// no rotation
IF ABS(angle)<g_smallAng THEN
	angle :=0;
	axis[1]:=1;
	axis[2]:=0;
	axis[3]:=0;
// rotate pi
ELSIF ABS(angle-pi)< g_smallAng THEN
	angle :=PI;
	axis[1]:=SQRT((LIMIT(-1, rot[1,1],1)+1)/2);
	axis[2]:=SQRT((LIMIT(-1, rot[2,2],1)+1)/2);
	axis[3]:=SQRT((limit(-1, rot[3,3],1)+1)/2);
	IF axis[1]>g_smallNum THEN
		axis[2]:=0.5*rot[1,2]/axis[1];
		axis[3]:=0.5*rot[1,3]/axis[1];
	ELSIF axis[2]>g_smallNum THEN
		axis[1]:=0.5*rot[2,1]/axis[2];
		axis[3]:=0.5*rot[2,3]/axis[2];
	ELSE
		axis[1]:=0.5*rot[3,1]/axis[3];
		axis[2]:=0.5*rot[3,2]/axis[3];
	END_IF
// others
ELSE
	tmp:=2*SIN(angle);
	axis[1]:=(rot[3,2]-rot[2,3])/tmp;
	axis[2]:=(rot[1,3]-rot[3,1])/tmp;
	axis[3]:=(rot[2,1]-rot[1,2])/tmp;
END_IF

// normalize
normalize(axis);

END_FUNCTION

// ---- AgiMaths/MatrixLib/normalize.TcPOU
// normalize the input vector
FUNCTION normalize : bool
VAR_IN_OUT
	vec :ARRAY[*] OF LREAL;
END_VAR
VAR
	m,i:DINT;
	vecNorm :LREAL;
END_VAR

m:=UPPER_BOUND(vec,1);
vecNorm :=norm(vec);

// if vector close to zero, remain the same;
IF vecNorm< g_smallNum THEN
	normalize :=FALSE;
	RETURN;
END_IF

FOR i:=1 TO m DO
	vec[i] := vec[i]/vecNorm;
END_FOR
normalize :=TRUE;

END_FUNCTION

// ---- AgiMaths/MatrixLib/norm.TcPOU
// return the norm of a vector
FUNCTION norm : LREAL
VAR_IN_OUT CONSTANT
	vec :ARRAY[*] OF LREAL;
END_VAR
VAR
	m,i:DINT;
END_VAR

m:=UPPER_BOUND(vec,1);
norm:=0;
FOR i:=1 TO m DO
	norm := norm + vec[i]*vec[i];
END_FOR

norm := SQRT(norm);

END_FUNCTION

// ---- AgiMaths/MatrixLib/vecMultiNum.TcPOU
// vecB=VecA*num
FUNCTION vecMultiNum : BOOL
VAR_IN_OUT CONSTANT
	vecA :ARRAY[*] OF LREAL;
END_VAR

VAR_INPUT
	num :LREAL;
END_VAR

VAR_IN_OUT
	vecB : ARRAY[*] OF LREAL;
END_VAR
VAR
	m :DINT;
	i :DINT;
END_VAR

m:=UPPER_BOUND(vecA,1);

FOR i:=1 TO m DO
		vecB[i]:=num*vecA[i];
END_FOR

END_FUNCTION

// ---- Mains/SlaveArmControl.TcPOU
PROGRAM SlaveArmControl
VAR
	// master robot data, input from master controller box
	m_masterRobotData AT %I* : MSCommu_MasterStatus;
	
	// all data from other tasks and controller 
	m_slaveInputDataPool : ST_SlaveInputDataPool;
		
	// slave robot data, ouput to master controller box
	m_slaveRobotData AT %Q* :MSCommu_slaveStatus;
	
	// slave robot status, including arm status and cartesian data, output to other tasks
	m_slaveStatus AT%Q* :ST_slaveStatus;
	
	// slave robot joint data, output to other tasks
	m_slaveJointsData AT %Q* :ST_slaveJointData;
	
	// flag to init robot
	m_robotInit :BOOL :=FALSE;
	
	// wait time before robot init  for ethercat to be statble 
	m_robotInitWaitTime : LREAL:=0;
	
	// slave robot
	m_slaveRobot:FB_SlaveRobot;

	// code execute time measure
	m_codeTime : Profiler;
	
END_VAR

m_codeTime(START:=TRUE, RESET:=TRUE);

// wait communication to be stable
IF(m_robotInitWaitTime<g_robotInitWaitTime) THEN
	m_robotInitWaitTime := m_robotInitWaitTime+g_slaveArmCtrlCycleTime;
	RETURN;
END_IF

// robot init
IF m_robotInit =FALSE THEN
	m_slaveRobot.Init();
	m_robotInit:=TRUE;
END_IF

// input from UI
UIInputProcess();

// master input data cast
masterInputDataCast(m_masterRobotData, m_slaveInputDataPool.m_masterStatus);

// robot run
m_slaveRobot.run(m_slaveInputDataPool);

// update data pool
m_slaveRobot.getStatus(m_slaveStatus,m_slaveJointsData);

// slave output data cast
slaveOutputDataCast(m_slaveInputDataPool.m_setupStatus, m_slaveStatus, m_slaveRobotData);

// output to UI
UIOutputProcess();

m_codeTime(START:=FALSE);

// convert from MSCommu_Mastertatus for master-slave communication to local ST_MasterStatus for control
METHOD masterInputDataCast : BOOL
VAR_IN_OUT CONSTANT
	masterInputData:MSCommu_MasterStatus;
END_VAR
VAR_IN_OUT
	masterStatus :ST_MasterStatus;
END_VAR

VAR
	i : INT;
END_VAR
masterStatus.m_masterHeartBeat := masterInputData.m_heartBeat;
masterStatus.m_motionScale := masterInputData.m_motionScale;
masterStatus.m_slaveSelfCheckFlag := masterInputData.m_slaveSelfCheckFlag OR GVL_interactUI.g_salveSelfCheckEnable;
masterStatus.m_masterStopButton := masterInputData.m_masterStopButton;
masterStatus.m_uiResetFault := masterInputData.m_uiResetFault;

FOR i:=1 TO g_mArmNum DO
	masterStatus.m_armState[i] := masterInputData.m_armState[i];
	masterStatus.m_teleSlaveArmIdx[i] :=masterInputData.m_teleSlaveArmIdx[i];
	masterStatus.m_gripAngle[i] := masterInputData.m_gripAngle[i];
	masterStatus.m_curArmPose[i].m_pos := masterInputData.m_curArmPose[i].m_pos;
	masterStatus.m_curArmPose[i].m_rot := masterInputData.m_curArmPose[i].m_rot;
	masterStatus.m_curArmTwist[i] :=masterInputData.m_curArmTwist[i];
	masterStatus.m_pedalHover[i] := masterInputData.m_pedalHover[i];
	masterStatus.m_electricKnifePedalTrigger[i] := masterInputData.m_electricKnifePedalTrigger[i];
	masterStatus.m_tryMSControl[i] := masterInputData.m_tryMSControl[i];
END_FOR
END_METHOD

// convert from local ST_SlaveStatus for control to MSCommu_SlaveStatus for master-slave communication
METHOD slaveOutputDataCast : BOOL
VAR_IN_OUT CONSTANT
	setupStatus :ST_SetupStatus;
	slaveStatus :ST_SlaveStatus;
END_VAR
VAR_IN_OUT 
	slaveOutputData : MSCommu_SlaveStatus;
END_VAR

VAR
	slavePoseInCart, slavePoseInScope:ST_Frame;
	tmpFrame :ST_Frame;
	i :INT;
END_VAR
// Slave heart beat
IF slaveOutputData.m_heartBeat > 10 THEN
	slaveOutputData.m_heartBeat :=0;
ELSE
	slaveOutputData.m_heartBeat :=slaveOutputData.m_heartBeat+1;
END_IF

FOR i := 1 TO g_sArmNum DO
	slaveOutputData.m_asepticDeployCompletedFlag :=SlaveArmControl.m_slaveInputDataPool.m_UIData.m_slaveArmDisableFlag[i] OR SlaveArmControl.m_slaveRobot.m_panelMountedFlag[i];	
	IF NOT slaveOutputData.m_asepticDeployCompletedFlag THEN
		EXIT;
	END_IF
END_FOR
IF slaveOutputData.m_asepticDeployCompletedFlag AND m_slaveInputDataPool.m_UIData.m_dumpEnergy < 30 THEN
	slaveOutputData.m_asepticDeployCompletedFlag := FALSE;
	FOR i:=1 TO g_sArmNum DO
		IF slaveStatus.m_armState[i] = SlaveArmState_MasterSlave THEN
			slaveOutputData.m_asepticDeployCompletedFlag := TRUE;
			EXIT;
		END_IF
	END_FOR
END_IF

slaveOutputData.m_seflCheckPass:=  m_slaveInputDataPool.m_UIData.m_armSelfCheckFinshed[1] AND  m_slaveInputDataPool.m_UIData.m_armSelfCheckFinshed[2] AND m_slaveInputDataPool.m_UIData.m_armSelfCheckFinshed[3] AND m_slaveInputDataPool.m_UIData.m_armSelfCheckFinshed[4] ;
slaveOutputData.m_endoscopeMounted :=slaveStatus.m_endoscopeMounted;
slaveOutputData.m_endoscopePose.m_pos :=slaveStatus.m_endoscopePose.m_pos;
slaveOutputData.m_endoscopePose.m_rot :=slaveStatus.m_endoscopePose.m_rot;
slaveOutputData.m_slaveStopButton := NOT SafetyCheck.m_stopButton;

FOR i:= 1 TO g_sArmNum DO
	slaveOutputData.m_armState[i] := slaveStatus.m_armState[i];
	slaveOutputData.m_instruStauts[i].m_fingerAngle := slaveStatus.m_instruStauts[i].m_fingerAngle;
	slaveOutputData.m_instruStauts[i].m_ready := slaveStatus.m_instruStauts[i].m_ready;
	slaveOutputData.m_instruStauts[i].m_type := slaveStatus.m_instruStauts[i].m_type;
	slaveOutputData.m_instruEnergyType[i] := m_slaveRobot.m_slaveArms[i].m_instrument.instruTypeInfo.m_energyType;
	slavePoseInCart := transform(setupStatus.m_curEndPose[i], slaveStatus.m_curArmPose[i]);
	tmpFrame :=invFrame(slaveStatus.m_endoscopePose);
	slavePoseInScope := transform(tmpFrame, slavePoseInCart);
	slaveOutputData.m_curArmPose[i].m_pos :=slavePoseInScope.m_pos;
	slaveOutputData.m_curArmPose[i].m_rot :=slavePoseInScope.m_rot;
	slaveOutputData.m_masterSlavePoseError[i] :=slaveStatus.m_masterSlavePoseError[i];
END_FOR
END_METHOD

// tranform data from UI(global variable write by ADS) to ST_UIData
METHOD UIInputProcess : BOOL
VAR_INPUT
END_VAR
VAR
	i:int;
END_VAR
// arm disable
FOR i:=1 TO g_sArmNum DO 
	m_slaveInputDataPool.m_UIData.m_slaveArmDisableFlag[i]:= FALSE;
END_FOR
IF GVL_interactUI.g_armIsDisable >0 AND GVL_interactUI.g_armIsDisable<= g_sArmNum THEN
	m_slaveInputDataPool.m_UIData.m_slaveArmDisableFlag[GVL_interactUI.g_armIsDisable]:= TRUE;
END_IF

m_slaveInputDataPool.m_UIData.m_dumpEnergy := GVL_interactUI.g_dumpEnergyUPS;
END_METHOD

METHOD UIOutputProcess : BOOL
VAR_INPUT
END_VAR

VAR
	i , j: INT;
END_VAR

VAR_STAT
	m_instruUsageCountsLast : ARRAY [1..g_sArmNum] OF ULINT;
END_VAR
//endoscope type
IF m_slaveRobot.m_endoScopeType = EndoscopeType_0  THEN
	GVL_interactUI.g_scopeType:= 0;
ELSIF m_slaveRobot.m_endoScopeType = EndoscopeType_30  THEN
	GVL_interactUI.g_scopeType := 30;
END_IF

//arm state machine
GVL_interactUI.g_armStateMachine.m_stateMachineArm1:=m_slaveStatus.m_armState[1];
GVL_interactUI.g_armStateMachine.m_stateMachineArm2:=m_slaveStatus.m_armState[2];
GVL_interactUI.g_armStateMachine.m_stateMachineArm3:=m_slaveStatus.m_armState[3];
GVL_interactUI.g_armStateMachine.m_stateMachineArm4:=m_slaveStatus.m_armState[4];

//arm is adjustment state
FOR i := 1 TO g_sArmNum BY 1 DO
	IF m_slaveStatus.m_armState[i] = SlaveArmState_Adjust OR SetupArmControl.m_setupStatus.m_armState[i] = SetupArmState_ManualAdjust 
							OR SetupArmControl.m_setupStatus.m_armState[i] = SetupArmState_AutoAdjust THEN
		GVL_interactUI.g_armIsAdjustment[i] := 1;
	ELSE
		GVL_interactUI.g_armIsAdjustment[i] := 0;
	END_IF
END_FOR


//arm self check status
FOR i := 1 TO g_sArmNum DO
	m_slaveInputDataPool.m_UIData.m_armInSelfCheck[i] := m_slaveStatus.m_armState[i] = SlaveArmState_SelfCheck AND NOT m_slaveInputDataPool.m_UIData.m_slaveArmDisableFlag[i];
	m_slaveInputDataPool.m_UIData.m_armSelfCheckFinshed[i] := m_slaveStatus.m_selfCheckPass[i] OR m_slaveInputDataPool.m_UIData.m_slaveArmDisableFlag[i];
END_FOR

IF m_slaveInputDataPool.m_UIData.m_armInSelfCheck[1] OR m_slaveInputDataPool.m_UIData.m_armInSelfCheck[2] OR m_slaveInputDataPool.m_UIData.m_armInSelfCheck[3] OR m_slaveInputDataPool.m_UIData.m_armInSelfCheck[4] THEN
	GVL_interactUI.g_slaveSelfCheckStatus := 1;
ELSIF m_slaveInputDataPool.m_UIData.m_armSelfCheckFinshed[1] AND m_slaveInputDataPool.m_UIData.m_armSelfCheckFinshed[2] AND m_slaveInputDataPool.m_UIData.m_armSelfCheckFinshed[3] AND m_slaveInputDataPool.m_UIData.m_armSelfCheckFinshed[4] THEN
	GVL_interactUI.g_slaveSelfCheckStatus := 2;
ELSE
	GVL_interactUI.g_slaveSelfCheckStatus := 0;
END_IF

//instrument information export to UI
FOR i := 1 TO g_sArmNum DO
	GVL_interactUI.g_instruInformatiom[i].m_instruIsConnected:=m_slaveStatus.m_instruStauts[i].m_ready;
	GVL_interactUI.g_instruInformatiom[i].m_instruInMasterSlave := (m_slaveStatus.m_armState[i] = SlaveArmState_MasterSlave OR m_slaveStatus.m_armState[i] = SlaveArmState_EndoScope);
	IF m_slaveStatus.m_instruStauts[i].m_type = InstruType_Endoscope THEN
		GVL_interactUI.g_instruInformatiom[i].m_instruType := 4;
		GVL_interactUI.g_scopeGravityAngle := m_slaveRobot.m_slaveArms[i].curDHJntPos[4];
	ELSE
		GVL_interactUI.g_instruInformatiom[i].m_instruType := m_slaveRobot.m_slaveArms[i].m_instrument.instruTypeInfo.m_energyType;
	END_IF
	
	GVL_interactUI.g_instruInformatiom[i].m_armId := i;
	GVL_interactUI.g_instruInformatiom[i].m_instruSerialNum :=  m_slaveRobot.m_slaveArms[i].m_instrument.onChipData.m_InstruseriesNum;
	GVL_interactUI.g_instruInformatiom[i].m_instruID := m_slaveRobot.m_slaveArms[i].m_instrument.instruType;
	GVL_interactUI.g_instruInformatiom[i].m_nameEn := m_slaveRobot.m_slaveArms[i].m_instrument.instruTypeInfo.m_instruName;
	GVL_interactUI.g_instruInformatiom[i].m_nameCh := m_slaveRobot.m_slaveArms[i].m_instrument.instruTypeInfo.m_instruNameCH;
	
	//instrument pedal hover and pedal active
	GVL_interactUI.g_instruInformatiom[i].m_pedalHover:=FALSE;
	GVL_interactUI.g_instruInformatiom[i].m_pedalActive := 0;
	FOR j := 1 TO g_mArmNum BY 1 DO
		 IF  m_slaveInputDataPool.m_masterStatus.m_teleSlaveArmIdx[j] > 0 AND   m_slaveInputDataPool.m_masterStatus.m_teleSlaveArmIdx[j] <= 4  THEN
			IF m_slaveInputDataPool.m_masterStatus.m_pedalHover[j] = TRUE THEN
				GVL_interactUI.g_instruInformatiom[m_slaveInputDataPool.m_masterStatus.m_teleSlaveArmIdx[j]].m_pedalHover:=TRUE;
			ELSE
				GVL_interactUI.g_instruInformatiom[m_slaveInputDataPool.m_masterStatus.m_teleSlaveArmIdx[j]].m_pedalHover:=FALSE;
			END_IF
			
			IF m_slaveRobot.m_slaveArms[m_slaveInputDataPool.m_masterStatus.m_teleSlaveArmIdx[j]].m_instrument.instruTypeInfo.m_energyType > 0 THEN
				IF m_slaveInputDataPool.m_masterStatus.m_electricKnifePedalTrigger[j] = 1 THEN 
					GVL_interactUI.g_instruInformatiom[m_slaveInputDataPool.m_masterStatus.m_teleSlaveArmIdx[j]].m_pedalActive := 1;
				ELSIF m_slaveInputDataPool.m_masterStatus.m_electricKnifePedalTrigger[j] = 2 THEN 
					GVL_interactUI.g_instruInformatiom[m_slaveInputDataPool.m_masterStatus.m_teleSlaveArmIdx[j]].m_pedalActive := 2;
				END_IF
			END_IF
			
		END_IF
	END_FOR
	
	// instrument out-of-view information
	GVL_interactUI.g_instruInformatiom[i].m_instruPosX:=m_slaveInputDataPool.m_slaveDynaData.m_insruViewData[i][1];
	GVL_interactUI.g_instruInformatiom[i].m_instruPosY:=m_slaveInputDataPool.m_slaveDynaData.m_insruViewData[i][2];
	GVL_interactUI.g_instruInformatiom[i].m_instruPosZ:=m_slaveInputDataPool.m_slaveDynaData.m_insruViewData[i][3];
	
	//instrument number of  use
	IF m_slaveRobot.m_slaveArms[i].m_instrument.onChipData.m_InstruUsageCounts <> m_InstruUsageCountsLast[i] THEN
		GVL_interactUI.g_instruInformatiom[i].m_useLifeplc := ULINT_TO_UINT(m_slaveRobot.m_slaveArms[i].m_instrument.onChipData.m_InstruUsageCounts);
	END_IF
	m_InstruUsageCountsLast[i] :=m_slaveRobot.m_slaveArms[i].m_instrument.onChipData.m_InstruUsageCounts;
	
	//read-write instrument number of use
	m_slaveRobot.m_slaveArms[i].m_instrument.writeNumOfUseToChip(GVL_interactUI.g_instruInformatiom[i].m_useLifeplc + 1 =  GVL_interactUI.g_instruInformatiom[i].m_useLifeUi AND m_slaveRobot.m_slaveArms[i].m_instrument.onChipData.m_InstruReadSucceed, GVL_interactUI.g_instruInformatiom[i].m_useLifeUi);

	//intrument total number of use
	GVL_interactUI.g_instruInformatiom[i].m_instruTotalLife := m_slaveRobot.m_slaveArms[i].m_instrument.instruTypeInfo.m_maxUseNum;
	//The coordinates of the instrument relative to the endoscope for UI display
END_FOR
END_METHOD

END_PROGRAM

// ---- FBs_Robots/FB_SlaveRobot.TcPOU
FUNCTION_BLOCK FB_SlaveRobot
VAR_INPUT
END_VAR
VAR_OUTPUT
END_VAR
VAR
	// flag if robot self-check passed
	m_selfCheckPass :ARRAY[1..g_sArmNum] OF BOOL :=[4(false)];
	
	// flag if master are connected
	m_masterOnLine :BOOL :=FALSE;
	m_masterOnLineCheck :FB_masterConnectionCheck;
	
	// master-slave motion scale
	m_motionScale :LREAL;
	
	// index(0 to 4) of slave arm which is tele-linked to master arm
	m_teleSlaveArmIdx :ARRAY[1..g_mArmNum] OF E_MatchedSlaveArmIdx;
	
	// flag if endoscope is mounted
	m_endoscopeMounted :BOOL := FALSE;
	
	// endoscope pose in cart coordinate
	m_endoscopePose : ST_Frame;
	
	// endoscope type 
	m_endoscopeType : E_EndoscopeType:= EndoScopeType_30;
	m_lastEndoScopePostureRobot : E_EndoscopePosture:= EndoScopePosture_HeadDown;
	m_lastEndoScopePostureUI : E_EndoscopePosture:= EndoScopePosture_HeadDown;
	
	// slave arms, responsible for arm kinematic and control
	m_slaveArms :ARRAY[1..g_sArmNum] OF FB_SlaveArm;
	
	// arm state
	m_slaveArmState:ARRAY[1..g_sArmNum] OF E_SlaveArmState:=[4(E_SlaveArmState.SlaveArmState_Error)];
	m_lastSlaveArmState:ARRAY[1..g_sArmNum] OF E_SlaveArmState:=[4(E_SlaveArmState.SlaveArmState_Error)];
	m_nextSlaveArmState:ARRAY[1..g_sArmNum] OF E_SlaveArmState:=[4(E_SlaveArmState.SlaveArmState_Error)];
	
	// matched master arm state
	m_matchedMasterArmState :ARRAY[1..g_sArmNum] OF E_MasterArmState:=[4(E_MasterArmState.MasterArmState_Error)];
	
	// flag if panel and instrument mounted
	m_panelMountedFlag :ARRAY[1..g_sArmNum] OF BOOL :=[4(FALSE)];
	m_instrumentMountedFlag :ARRAY[1..g_sArmNum] OF BOOL :=[4(FALSE)];
	
	// flag if enable instrument invasion after it mounted
	m_instruInvasionEnableFlag :ARRAY[1..g_sArmNum] OF BOOL :=[4(FALSE)];
	
	// all arm controller instance 
	m_armCtrlFactory :ARRAY[1..g_sArmNum,1..SlaveArmState_totalNum] OF I_SlaveArmCtrl;
	m_armError :ARRAY[1..g_sArmNum] OF FB_SlaveCtrlError;
	m_armInit :ARRAY[1..g_sArmNum] OF FB_SlaveCtrlInit;
	m_armSelfCheck :ARRAY[1..g_sArmNum] OF FB_SlaveCtrlSelfCheck;
	m_armStandBy :ARRAY[1..g_sArmNum] OF FB_SlaveCtrlStandBy;
	m_mountPanel :ARRAY[1..g_sArmNum] OF FB_SlaveCtrlMountPanel;
	m_panelReady :ARRAY[1..g_sArmNum] OF FB_SlaveCtrlPanelReady;
	m_mountInstru :ARRAY[1..g_sArmNum] OF FB_SlaveCtrlMountInstru;
	m_instruReady :ARRAY[1..g_sArmNum] OF FB_SlaveCtrlInstruReady;
	m_armMasterSlave :ARRAY[1..g_sArmNum] OF FB_SlaveCtrlMasterSlave;
	m_scopeReady :ARRAY[1..g_sArmNum] OF FB_SlaveCtrlScopeReady;
	m_armEndoscope :ARRAY[1..g_sArmNum] OF FB_SlaveCtrlEndoscope;
	m_armAdjust :ARRAY[1..g_sArmNum] OF FB_SlaveCtrlAdjust;
	m_armPackage :ARRAY[1..g_sArmNum] OF FB_SlaveCtrlPackage;
	m_armCart :ARRAY[1..g_sArmNum] OF FB_SlaveCtrlCart;
	m_armGraCali :ARRAY[1..g_sArmNum] OF FB_SlaveCtrlGraCali;
	m_armTest :ARRAY[1..g_sArmNum] OF FB_SlaveCtrlTest;
	m_instruRetract :ARRAY[1..g_sArmNum] OF FB_SlaveCtrlInstruRetract;
	m_instruInvasion :ARRAY[1..g_sArmNum] OF FB_SlaveCtrlInstruInvasion;
	m_armDisable :ARRAY[1..g_sArmNum] OF FB_SlaveCtrlDisable;
	m_instruCali :ARRAY[1..g_sArmNum] OF FB_SlaveCtrlInstruCali;
	m_scopeToggle :ARRAY[1..g_sArmNum] OF FB_SlaveCtrlScopeToggle;
	m_Performance :ARRAY[1..g_sArmNum] OF FB_SlaveCtrlPerformance;
	m_armStop :ARRAY[1..g_sArmNum] OF FB_SlaveCtrlStop;
	
	// arm controller interface
	m_armCtrl :ARRAY[1..g_sArmNum] OF I_SlaveArmCtrl;
	m_armCtrlCmds :ARRAY[1..g_sArmNum] OF ST_SlaveArmCtrlCmds;

END_VAR

METHOD PROTECTED controllerTransit : BOOL
VAR_INPUT
END_VAR
VAR
	i:int;
END_VAR
FOR i:=1 TO g_sArmNum DO 
	// Controller transit
	IF m_nextSlaveArmState[i]<> m_slaveArmState[i] THEN
		// reset current controller
		m_armCtrl[i].reset();
		
		// transit to new controller
		m_lastSlaveArmState[i]:=m_slaveArmState[i];
		m_slaveArmState[i]:=m_nextSlaveArmState[i];
		m_armCtrl[i]:=m_armCtrlFactory[i,m_slaveArmState[i]];
		
		// init next controller
		m_armCtrl[i].Init(m_slaveArms[i],m_armCtrlCmds[i]);
		m_slaveArms[i].updateCmds(m_armCtrlCmds[i]);
	END_IF
END_FOR
END_METHOD

METHOD PUBLIC getStatus : BOOL
VAR_IN_OUT
	// slave robot information, including arm status and cartesian data
	r_slaveStatus :ST_SlaveStatus;
	
	// slave robot joint data
	r_slaveJointsData :ST_SlaveJointData;
	
END_VAR

VAR
	i:INT;
END_VAR
r_slaveStatus.m_armState:=m_slaveArmState;
r_slaveStatus.m_endoscopeMounted :=m_endoscopeMounted;
r_slaveStatus.m_endoscopePose :=m_endoscopePose;

FOR i:=1 TO g_sArmNum DO
	r_slaveStatus.m_selfCheckPass[i] := m_selfCheckPass[i];	

	// instrument data
	r_slaveStatus.m_instruStauts[i].m_type:=m_slaveArms[i].instrument.m_instruType;
	r_slaveStatus.m_instruStauts[i].m_ready:=m_instrumentMountedFlag[i];
	r_slaveStatus.m_instruStauts[i].m_fingerAngle:=m_slaveArms[i].curGripAngle;
	r_slaveStatus.m_instruReadErrId[i] := m_slaveArms[i].instrument.onChipData.m_ErrorID;
	r_slaveStatus.m_instruInstallStatus[i] := m_slaveArms[i].instruOn;
	r_slaveStatus.m_instruClampErrId[i] := m_mountInstru[i].instruClampErrId;
	r_slaveStatus.m_panelInstallStatus[i] := m_slaveArms[i].panelOn;
	r_slaveStatus.m_panelClampErrId[i] := m_mountPanel[i].panelClampErrId;
	r_slaveStatus.m_trocarOnFlag[i] := m_slaveArms[i].trocarOn;
	r_slaveStatus.m_masterOnLine := m_masterOnLine;
	// cartesion
	r_slaveStatus.m_curArmPose[i]:=m_slaveArms[i].curCartPose;
	r_slaveStatus.m_simArmPose[i]:=m_slaveArms[i].simCartPose;
	r_slaveStatus.m_masterSlavePoseError[i] := m_armMasterSlave[i].masterSlavePoseErr;
	// joint
	r_slaveJointsData.m_curMotorPos[i]:=m_slaveArms[i].curMotorPos;
	r_slaveJointsData.m_curLinkPos[i]:=m_slaveArms[i].curLinkPos;
	r_slaveJointsData.m_curJntPos[i]:=m_slaveArms[i].curJntPos;
	r_slaveJointsData.m_curJntVel[i]:=m_slaveArms[i].curJntVel;
	r_slaveJointsData.m_curDHJntPos[i]:=m_slaveArms[i].curDHJntPos;
	
	// command info
	// cartesion
	r_slaveStatus.m_cmdArmPose[i]:=m_slaveArms[i].cmdCartPose;
	// joint info
	r_slaveJointsData.m_cmdJntPos[i]:=m_slaveArms[i].cmdJntPos;
	
END_FOR
END_METHOD

METHOD PUBLIC Init : BOOL
VAR_INPUT
END_VAR
VAR
	i:INT;
END_VAR
FOR i:=1 TO g_sArmNum DO
	// arm init
	m_slaveArms[i].Init(i);
	m_slaveArmState[i]:=SlaveArmState_Init;
	m_lastSlaveArmState[i]:=SlaveArmState_Init;
	m_nextSlaveArmState[i]:=SlaveArmState_Init;
	m_selfCheckPass[i]:=false;
	
	// command init
	m_armCtrlCmds[i].m_jntEnableFlag := g_zeroVec8i;
	m_armCtrlCmds[i].m_jntOPMode := g_slaveAllPosMode;
	m_armCtrlCmds[i].m_cmdCartPose := m_slaveArms[i].curCartPose;
	m_armCtrlCmds[i].m_cmdCartTwist := g_zeroVec6d;
	m_armCtrlCmds[i].m_cmdJntPos := m_slaveArms[i].curJntPos;
	m_armCtrlCmds[i].m_cmdJntVel := g_zeroVec8d;
	m_armCtrlCmds[i].m_cmdJntAcc := g_zeroVec8d;
	m_armCtrlCmds[i].m_cmdJntTrq := g_zeroVec8d;
	
	// generate controller factory
	m_armCtrlFactory[i,SlaveArmState_Error] := m_armError[i];
	m_armCtrlFactory[i,SlaveArmState_Init] := m_armInit[i];
	m_armCtrlFactory[i,SlaveArmState_SelfCheck] := m_armSelfCheck[i];
	m_armCtrlFactory[i,SlaveArmState_Standby] := m_armStandBy[i];
	m_armCtrlFactory[i,SlaveArmState_MountPanel] := m_mountPanel[i];
	m_armCtrlFactory[i,SlaveArmState_PanelReady] := m_panelReady[i];
	m_armCtrlFactory[i,SlaveArmState_MountInstru] := m_mountInstru[i];
	m_armCtrlFactory[i,SlaveArmState_InstruReady] := m_instruReady[i];
	m_armCtrlFactory[i,SlaveArmState_MasterSlave] := m_armMasterSlave[i];
	m_armCtrlFactory[i,SlaveArmState_ScopeReady] := m_scopeReady[i];
	m_armCtrlFactory[i,SlaveArmState_EndoScope] := m_armEndoscope[i];
	m_armCtrlFactory[i,SlaveArmState_Adjust] := m_armAdjust[i];
	m_armCtrlFactory[i,SlaveArmState_Package] := m_armPackage[i];
	m_armCtrlFactory[i,SlaveArmState_Cart] := m_armCart[i];
	m_armCtrlFactory[i,SlaveArmState_GravityCali] := m_armGraCali[i];
	m_armCtrlFactory[i,SlaveArmState_Test] := m_armTest[i];
	m_armCtrlFactory[i,SlaveArmState_InstruRetract] := m_instruRetract[i];
	m_armCtrlFactory[i,SlaveArmState_InstruInvasion] := m_instruInvasion[i];
	m_armCtrlFactory[i,SlaveArmState_Disable] := m_armDisable[i];
	m_armCtrlFactory[i,SlaveArmState_InstruCali] := m_instruCali[i];
	m_armCtrlFactory[i,SlaveArmState_ScopeToggle] := m_scopeToggle[i];
	m_armCtrlFactory[i,SlaveArmState_Performance] := m_Performance[i];
	m_armCtrlFactory[i,SlaveArmState_Stop] := m_armStop[i];
	
	// assign controller
	m_armCtrl[i]:=m_armCtrlFactory[i,m_slaveArmState[i]];
	m_armCtrl[i].Init(m_slaveArms[i],m_armCtrlCmds[i]);
END_FOR
END_METHOD

METHOD PUBLIC run : BOOL
VAR_IN_OUT CONSTANT
	i_slaveInputDataPool:ST_SlaveInputDataPool;
END_VAR
VAR
	i:INT;
END_VAR
m_motionScale := i_slaveInputDataPool.m_masterStatus.m_motionScale;
m_teleSlaveArmIdx := i_slaveInputDataPool.m_masterStatus.m_teleSlaveArmIdx;

// check master connection
m_masterOnLine := m_masterOnLineCheck.check(i_slaveInputDataPool.m_masterStatus.m_masterHeartBeat);

// check if endoscope is mounted
m_endoscopeMounted := FALSE;
FOR i:=1 TO g_sArmNum DO 
	IF m_slaveArms[i].instrument.m_instruType=InstruType_endoscope THEN
		m_endoscopeMounted := TRUE;
		m_endoscopePose := transform(i_slaveInputDataPool.m_setupStatus.m_curEndPose[i], m_slaveArms[i].curCartPose);
		m_endoScopeType := m_slaveArms[i].instrument.curScopeType;
		
		//set endoscope  posture from UI data
		updateScopeUIInfo();
	END_IF
END_FOR

// update arm status
FOR i:=1 TO g_sArmNum DO
	// update dynamic data
	m_slaveArms[i].updateDyna(i_slaveInputDataPool.m_slaveDynaData);
								
	// update slave arm kinematics
	m_slaveArms[i].updateStatus();
END_FOR

// state machine transition
stateMachine(i_slaveInputDataPool);

// controller transition
controllerTransit();

// run arm controller
FOR i:=1 TO g_sArmNum DO
	// null ptr check
	ASSERT(0 <> m_armCtrl[i]);
	
	// run controller
	m_armCtrl[i].run(m_endoscopePose, i_slaveInputDataPool.m_MasterStatus,
					i_slaveInputDataPool.m_setupStatus, m_SlaveArms[i],m_armCtrlCmds[i]);

	// update commands to drivers
	m_slaveArms[i].updateCmds(m_armCtrlCmds[i]);
END_FOR
END_METHOD

// state machine check and transit 
METHOD PROTECTED stateMachine : BOOL
VAR_IN_OUT CONSTANT
		i_slavesInputDataPool:ST_SlaveInputDataPool;
END_VAR
VAR
	i,j:INT;
	potentGripTrig :BOOL;
END_VAR
// check instrument state
FOR i:=1 TO g_sArmNum DO
	// statues check
	IF m_slaveArms[i].panelOn = FALSE THEN
		m_panelMountedFlag[i]:=FALSE;
	END_IF
	IF m_slaveArms[i].instruOn = FALSE THEN
		m_instrumentMountedFlag[i]:=FALSE;
		// clear instrument control backlash
		m_slaveArms[i].instruJntBacklash:=g_zeroVec5d;		
		m_armMasterSlave[i].clearBacklash();
	END_IF
END_FOR

// get matched master arm state
FOR i:=1 TO g_sArmNum DO 
	m_matchedMasterArmState[i]:=MasterArmState_Error;
	FOR j:=1 TO g_mArmNum DO 
		IF i = i_slavesInputDataPool.m_masterStatus.m_teleSlaveArmIdx[j] THEN
			m_matchedMasterArmState[i] := i_slavesInputDataPool.m_masterStatus.m_armState[j];
		END_IF
	END_FOR
END_FOR

// check if to enable instrument invasion 
FOR i:=1 TO g_sArmNum DO
	IF SlaveArmState_Adjust = m_slaveArmState[i] OR SlaveArmState_Cart = m_slaveArmState[i] OR i_slavesInputDataPool.m_setupStatus.m_armState[i] = SetupArmState_ManualAdjust OR
	    m_slaveArms[i].instrument.instruType = InstruType_Endoscope	 THEN
		m_instruInvasionEnableFlag[i]:=FALSE;
		m_slaveArms[i].resetInstruDepth();
	ELSIF m_instrumentMountedFlag[i] AND m_slaveArms[i].instrument.instruType <> InstruType_Endoscope AND m_slaveArmState[i] <> SlaveArmState_InstruInvasion THEN
		m_instruInvasionEnableFlag[i]:=TRUE;
		m_slaveArms[i].setInstruDepth();
	END_IF
END_FOR  

// state machine transit
FOR i:=1 TO g_sArmNum DO
	CASE m_slaveArmState[i] OF
		// error
		SlaveArmState_Error:
			IF FALSE = i_slavesInputDataPool.m_safetyData.m_slaveErrFlag[i] THEN
				// to standby
				IF m_selfCheckPass[i] THEN
					m_nextSlaveArmState[i] :=SlaveArmState_Standby;
				// to init
				ELSE
					m_nextSlaveArmState[i] :=SlaveArmState_Init;
				END_IF
			END_IF
			// to adjust
			IF (m_slaveArms[i].adjustOn) THEN
				m_nextSlaveArmState[i]:=SlaveArmState_Adjust;
			END_IF
			
		// init
		SlaveArmState_Init:
			m_selfCheckPass[i]:=FALSE;
			m_slaveArms[i].instrument.resetArmLED :=TRUE;
			// to selfcheck
			IF m_armCtrl[i].isFinished AND i_slavesInputDataPool.m_masterStatus.m_slaveSelfCheckFlag  THEN
				m_nextSlaveArmState[i]:=SlaveArmState_SelfCheck;
			// to adjust
			ELSIF m_slaveArms[i].adjustOn THEN
				m_nextSlaveArmState[i]:=SlaveArmState_Adjust;
			END_IF

		//self check
		SlaveArmState_SelfCheck:
			// to standby
			IF m_armCtrl[i].isFinished  THEN
				m_nextSlaveArmState[i]:=SlaveArmState_Standby;
				m_selfCheckPass[i]:=TRUE;
			END_IF
		
		//standby
		SlaveArmState_Standby:
			// to mount panel
			IF m_slaveArms[i].panelOn THEN 
				IF m_panelMountedFlag[i] THEN
					m_nextSlaveArmState[i]:=SlaveArmState_PanelReady;
				ELSE
					m_nextSlaveArmState[i]:=SlaveArmState_MountPanel;
				END_IF
			// to adjust
			ELSIF m_slaveArms[i].adjustOn THEN
				m_nextSlaveArmState[i]:=SlaveArmState_Adjust;
			END_IF
		
		//mount panel
		SlaveArmState_MountPanel:
			// to panel ready
			IF m_armCtrl[i]. isFinished THEN
				m_nextSlaveArmState[i]:=SlaveArmState_PanelReady;
				m_panelMountedFlag[i] :=TRUE;
				
			// to standby
			ELSIF NOT(m_slaveArms[i].panelOn) THEN
				m_nextSlaveArmState[i]:=SlaveArmState_Standby;
			END_IF
		
		//panel ready
		SlaveArmState_PanelReady:
			// to adjust
			IF (m_slaveArms[i].adjustOn) THEN
				m_nextSlaveArmState[i]:=SlaveArmState_Adjust;
			// to stand by
			ELSIF NOT(m_slaveArms[i].panelOn) THEN
				m_nextSlaveArmState[i]:=SlaveArmState_Standby;
			ELSIF m_slaveArms[i].instruOn   THEN
				IF m_instrumentMountedFlag[i] THEN
					// to scope ready
					IF  InstruType_endoscope = m_slaveArms[i].instrument.m_instruType AND m_slaveArms[i].instruReady() THEN 
						m_nextSlaveArmState[i]:=SlaveArmState_ScopeReady;
					// to scope toggle
					ELSIF  InstruType_endoscope = m_slaveArms[i].instrument.m_instruType AND 
								(m_slaveArms[i].instrument.curScopePosture <> m_slaveArms[i].instrument.nextScopePosture OR
								m_slaveArms[i].instrument.curScopeType <> m_slaveArms[i].instrument.nextScopeType) THEN
						m_nextSlaveArmState[i] := SlaveArmState_ScopeToggle;
					// to instrument ready
					ELSIF  m_slaveArms[i].instruReady() THEN
						m_nextSlaveArmState[i]:=SlaveArmState_InstruReady;
					END_IF
				// to mount instrument/endoscope
				ELSIF m_slaveArms[i].readyForInstruMount() THEN
					m_nextSlaveArmState[i]:=SlaveArmState_MountInstru;
				END_IF
			// to instrument retract
			ELSIF  NOT(m_slaveArms[i].readyForInstruMount())  THEN
				m_nextSlaveArmState[i]:=SlaveArmState_InstruRetract;
			END_IF
			
		//mount instrument
		SlaveArmState_MountInstru:
			// to panel ready
			IF NOT(m_slaveArms[i].instruOn)  THEN
				m_nextSlaveArmState[i]:=SlaveArmState_PanelReady;
			ELSIF m_armCtrl[i].isFinished THEN
				m_instrumentMountedFlag[i] :=TRUE;
				
				// to instrument invasion
				IF m_instruInvasionEnableFlag[i] THEN
					m_nextSlaveArmState[i] := SlaveArmState_InstruInvasion;
				// to panel ready
				ELSE
					m_nextSlaveArmState[i]:=SlaveArmState_PanelReady;
				END_IF
				
			END_IF
		
		// instrument ready
		SlaveArmState_InstruReady:
			// to instrument retract
			IF  NOT(m_slaveArms[i].instruOn)  THEN
				m_nextSlaveArmState[i]:=SlaveArmState_InstruRetract;
			// to Adjust
			ELSIF (m_slaveArms[i].adjustOn) THEN
				m_nextSlaveArmState[i]:=SlaveArmState_Adjust;
			// to master-slave
			ELSIF MasterArmState_MasterSlave = m_matchedMasterArmState[i] THEN
				m_nextSlaveArmState[i] := SlaveArmState_MasterSlave;
			END_IF
		
		//master slave control
		SlaveArmState_MasterSlave:
			m_slaveArms[i].instruJntBacklash :=  m_armMasterSlave[i].InstruBacklash;
			// to Adjust
			IF (m_slaveArms[i].adjustOn) THEN
				m_nextSlaveArmState[i]:=SlaveArmState_Adjust;
			// to stop
			ELSIF MasterArmState_MasterSlave <> m_matchedMasterArmState[i] OR m_armCtrl[i].isFinished THEN
				m_nextSlaveArmState[i]:=SlaveArmState_Stop;
			// to instrument retract
			ELSIF  NOT(m_slaveArms[i].panelOn) OR NOT(m_slaveArms[i].instruOn) THEN
				m_nextSlaveArmState[i]:=SlaveArmState_InstruRetract;
			END_IF
		
		//endoscope ready
		SlaveArmState_ScopeReady:
			// to instrument retract
			IF NOT(m_slaveArms[i].instruOn) THEN
				m_nextSlaveArmState[i]:=SlaveArmState_InstruRetract;
			// to Adjust
			ELSIF (m_slaveArms[i].adjustOn) THEN
				m_nextSlaveArmState[i]:=SlaveArmState_Adjust;
			// to scope toggle
			ELSIF m_slaveArms[i].instrument.curScopePosture <> m_slaveArms[i].instrument.nextScopePosture OR
					m_slaveArms[i].instrument.curScopeType <> m_slaveArms[i].instrument.nextScopeType THEN
				m_nextSlaveArmState[i] := SlaveArmState_ScopeToggle;
			// to endoscope control
			ELSIF MasterArmState_Endoscope = i_slavesInputDataPool.m_masterStatus.m_armState[1] AND 
				  MasterArmState_Endoscope = i_slavesInputDataPool.m_masterStatus.m_armState[2] THEN
				m_nextSlaveArmState[i] := SlaveArmState_EndoScope;
			END_IF
		
		//endoscope control
		SlaveArmState_EndoScope:
			// to Adjust
			IF (m_slaveArms[i].adjustOn) THEN
				m_nextSlaveArmState[i]:=SlaveArmState_Adjust;
			// to stop
			ELSIF MasterArmState_Endoscope <> i_slavesInputDataPool.m_masterStatus.m_armState[1]
				OR MasterArmState_Endoscope <> i_slavesInputDataPool.m_masterStatus.m_armState[2] THEN
				m_nextSlaveArmState[i]:=SlaveArmState_Stop;
			// to scope toggle
			ELSIF m_slaveArms[i].instrument.curScopePosture <> m_slaveArms[i].instrument.nextScopePosture OR
					m_slaveArms[i].instrument.curScopeType <> m_slaveArms[i].instrument.nextScopeType THEN
				m_nextSlaveArmState[i] := SlaveArmState_ScopeToggle;
			// to instrument retract
			ELSIF  NOT(m_slaveArms[i].panelOn) OR NOT(m_slaveArms[i].instruOn) THEN
				m_nextSlaveArmState[i]:=SlaveArmState_InstruRetract;
			END_IF
			
		//arm adjust
		SlaveArmState_Adjust:
			IF m_slaveArms[i].adjustFallEdge AND m_armCtrl[i].timePeriod > 0.25 THEN
				// to init
				IF NOT (m_selfCheckPass[i]) THEN
					m_nextSlaveArmState[i] :=SlaveArmState_Init;
				// to standby
				ELSE
					m_nextSlaveArmState[i] :=SlaveArmState_Standby;
				END_IF
			END_IF
		
		//scope toggle
		SlaveArmState_ScopeToggle:
			// to instrument retract
			IF NOT(m_slaveArms[i].instruOn) THEN
				m_nextSlaveArmState[i]:=SlaveArmState_InstruRetract;
			// to standby
			ELSIF m_armCtrl[i].isFinished THEN
				m_nextSlaveArmState[i] :=SlaveArmState_Standby;
			END_IF
		
		// package
		SlaveArmState_Package:
			// to Adjust
			IF (m_slaveArms[i].adjustOn) THEN
				m_nextSlaveArmState[i]:=SlaveArmState_Adjust;
			// to standby
			ELSIF m_armCtrl[i].isFinished THEN
				m_nextSlaveArmState[i]:=SlaveArmState_Standby;
			END_IF
			
		// Cart
		SlaveArmState_Cart:
		
		// Gravity Calibration
		SlaveArmState_GravityCali:
			// to Adjust
			IF (m_slaveArms[i].adjustOn) THEN
				m_nextSlaveArmState[i]:=SlaveArmState_Adjust;
			// to standby
			ELSIF m_armCtrl[i].isFinished THEN
				m_nextSlaveArmState[i]:=SlaveArmState_Standby;
			END_IF
			
		//arm test
		SlaveArmState_Test:
			// to stop
			IF  m_armCtrl[i].isFinished THEN
				m_nextSlaveArmState[i]:=SlaveArmState_Stop;
			END_IF
		
		//arm Performance
		SlaveArmState_Performance:
			// to standby
			IF  m_armCtrl[i].isFinished THEN
				m_nextSlaveArmState[i]:=SlaveArmState_Standby;
			END_IF		
			
		//arm stop
		SlaveArmState_Stop:
			// to standby
			IF  m_armCtrl[i].isFinished THEN
				m_nextSlaveArmState[i]:=SlaveArmState_Standby;
			END_IF
		
		// instrument retract
		SlaveArmState_InstruRetract:
			// to Adjust
			IF (m_slaveArms[i].adjustOn) THEN
				m_nextSlaveArmState[i]:=SlaveArmState_Adjust;
			// to standby
			ELSIF m_armCtrl[i].isFinished THEN
				m_nextSlaveArmState[i]:=SlaveArmState_Standby;
			END_IF
		
		// instrument invasion
		SlaveArmState_InstruInvasion:
			// to instrument retract
			IF NOT m_slaveArms[i].instruOn THEN
				m_nextSlaveArmState[i]:=SlaveArmState_InstruRetract;
			// to Adjust
			elsIF (m_slaveArms[i].adjustOn) THEN
				m_nextSlaveArmState[i]:=SlaveArmState_Adjust;
			// to instrument ready
			ELSIF m_armCtrl[i].isFinished THEN
			// to panel ready
				m_nextSlaveArmState[i]:=SlaveArmState_PanelReady;
			END_IF
		
		// arm disable
		SlaveArmState_Disable:
			IF NOT(i_slavesInputDataPool.m_UIData.m_slaveArmDisableFlag[i]) THEN
				// to standby
				IF m_selfCheckPass[i] THEN
					m_nextSlaveArmState[i] :=SlaveArmState_Standby;
				// to init
				ELSE
					m_nextSlaveArmState[i] :=SlaveArmState_Init;
				END_IF
			END_IF
	END_CASE
	
	// control is forbidden if setup arm is not in Hold
	IF SetupArmState_Hold <> i_slavesInputDataPool.m_setupStatus.m_armState[i] AND
		(SlaveArmState_InstruReady = m_nextSlaveArmState[i] OR SlaveArmState_MasterSlave = m_nextSlaveArmState[i]
		 OR SlaveArmState_ScopeReady = m_nextSlaveArmState[i] OR SlaveArmState_EndoScope = m_nextSlaveArmState[i]) THEN
		m_nextSlaveArmState[i]:=SlaveArmState_Standby;
	END_IF
	
	// arm disable
	IF i_slavesInputDataPool.m_UIData.m_slaveArmDisableFlag[i] THEN
		m_nextSlaveArmState[i] := SlaveArmState_Disable;
	// error check
	ELSIF i_slavesInputDataPool.m_safetyData.m_slaveErrFlag[i] AND NOT m_slaveArms[i].adjustOn THEN
		m_nextSlaveArmState[i]:=SlaveArmState_Error;
	END_IF
END_FOR
END_METHOD

METHOD PROTECTED updateScopeUIInfo : BOOL
VAR_INPUT
END_VAR
VAR
	i:INT;
END_VAR
// check if endoscope is mounted
FOR i:=1 TO g_sArmNum DO 
	IF m_slaveArms[i].instrument.m_instruType=InstruType_endoscope THEN
		
		// update command endoscope posture from UI
		IF GVL_interactUI.g_scopeUpDown <> m_lastEndoScopePostureUI AND m_slaveArms[i].instrument.curScopeType = EndoScopeType_30 THEN
			IF GVL_interactUI.g_scopeUpDown = 1 THEN
				m_slaveArms[i].instrument.nextScopePosture := EndoScopePosture_HeadDown;
			ELSIF  GVL_interactUI.g_scopeUpDown = 2 THEN
				m_slaveArms[i].instrument.nextScopePosture := EndoscopePosture_HeadUp;
			END_IF
		END_IF
		
		// update current endoscope posture to UI
		IF m_slaveArms[i].instrument.curScopePosture <> m_lastEndoScopePostureRobot THEN
			IF m_slaveArms[i].instrument.curScopePosture = EndoScopePosture_HeadDown THEN
				GVL_interactUI.g_scopeUpDown := 1 ;
			ELSIF  m_slaveArms[i].instrument.curScopePosture = EndoScopePosture_HeadUp THEN
				GVL_interactUI.g_scopeUpDown := 2;
			END_IF
		END_IF
		m_lastEndoScopePostureRobot := m_slaveArms[i].instrument.curScopePosture;
		
	END_IF
END_FOR

m_lastEndoScopePostureUI := GVL_interactUI.g_scopeUpDown;
END_METHOD

END_FUNCTION_BLOCK

// ---- FBs_Auxiliary/FB_masterConnectionCheck.TcPOU
FUNCTION_BLOCK FB_masterConnectionCheck
VAR
	// current state 
	m_isConnected :BOOL :=FALSE;
	
	// last heart beat
	m_lastHeartBeat :INT:=0 ;
	
	// current conneciton cycles
	m_curConnectionCycles :INT:=0;
	
	// current disconneciton cycles
	m_curDisconnectionCycles :INT:=0;
	
	// conneciton cycles thresshold
	m_connectionCyclesThres :INT:=5;
	
END_VAR

METHOD PUBLIC check : BOOL
VAR_INPUT
	i_heartBeat :INT;
END_VAR
// current is disconnected
IF NOT(m_isConnected) THEN
	m_curDisconnectionCycles:=0;
	
	IF  i_heartBeat <> m_lastHeartBeat THEN
		m_curConnectionCycles :=  m_curConnectionCycles +1;
	ELSE
		m_curConnectionCycles :=0;
	END_IF
	
	IF  m_curConnectionCycles >= m_connectionCyclesThres THEN
		m_isConnected := TRUE;
	END_IF

// current is connected
ELSE
	m_curConnectionCycles :=0;
	
	IF  i_heartBeat = m_lastHeartBeat THEN
		m_curDisconnectionCycles := m_curDisconnectionCycles +1;
	ELSE
		m_curDisconnectionCycles :=0;
	END_IF
	
	IF m_curDisconnectionCycles>= m_connectionCyclesThres THEN
		m_isConnected:=FALSE;
	END_IF

END_IF

m_lastHeartBeat:= i_heartBeat;
check:=m_isConnected;
END_METHOD

END_FUNCTION_BLOCK

// ---- FBs_Robots/FB_SlaveArm.TcPOU
FUNCTION_BLOCK FB_SlaveArm
VAR_INPUT
END_VAR
VAR_OUTPUT
END_VAR
VAR
	// arm index, from 1 to 4
	m_armIdx: INT;
	
	// joints
	m_joints :ARRAY[1..g_sJntNum] OF FB_SlaveJoint;
	
	//  panel and insturment detect
	m_panelInstrumentOnIO AT%I*	:UDINT;
	m_panelDetect :FB_PanelDetect;
	m_instruDetect :FB_InstrumentDetect;
	m_instruNearDetect :FB_InstruNearDetect;
	m_panelOnFlag :BOOL:=FALSE;
	m_instruOnFlag :BOOL:=FALSE;
	m_instruNearFlag :BOOL:=FALSE;

	
	// trocar and  adjust detect
	m_adjustIO AT%I* :UDINT;
	m_adjustDetect :FB_AdjustDetect;
	m_trocarDetect : FB_TrocarDetect;
	m_adjustOnFlag :BOOL;
	m_trocarOnFlag :BOOL :=FALSE;
	m_adjustFallEdge :BOOL:=false;
	m_adjustFallEdgeDetect : F_TRIG;
	
	//endoscope type and posture switch
	m_endoscopeTypeSwitch : FB_IOToggleCheck;
	m_endoscopePostureSwitch : FB_IOToggleCheck;
	
	// instrument instance
	m_instrument : FB_Instrument;
	
	// instrument invasion depth before it's unmounted
	m_instruInvasionDepth :LREAL;

	// arm cartesian data, defined in each arm origin
	m_curCartPose	:ST_Frame;
	m_curCartTwist: Vec6d;
	m_cmdCartTwist :Vec6d;
	m_cmdCartPose:ST_Frame;
	
	// arm joint data
	m_curMotorPos :Vec8d;
	m_curLinkPos :Vec8d;
	m_curLinkSingle :Vec8d;
	m_curJntPos :Vec8d;
	m_curDHJntPos :Vec6d;
	m_curGripAngle :LREAL;
	m_curJntVel :Vec8d;
	m_curDHJntVel :Vec6d;
	m_curJntTrq :Vec8d;
	m_rawJntCurrent :Vec8d;
	m_filtJntCurrent :Vec8d;
	m_cmdJntTrq :Vec8d;
	m_cmdJntCurrent : Vec8d;
	m_cmdJntPos :Vec8d;
	m_cmdJntVel :Vec8d;
	
	// intrument joint backlash
	m_instruJntBacklash :Vec5d:=g_zeroVec5d;
		
	// arm dynamic data
	m_jntGravity : Vec8d:=g_zeroVec8d;
	m_jntMassMat : Mat3d;
	
	// arm jacobian and inverse
	m_jaco : Mat6d;
	
	// simulated status
	m_simJntPos :Vec8d;
	m_simDHJntPos :Vec6d;
	m_simGripAngle :LREAL;
	m_simCartPose : ST_Frame;
	m_simJaco : Mat6d;
	m_simJacoInv :Mat6d;
	m_isSingularity:BOOL:=false;
	
	// joint position controller
	m_jntPIDCtrl :ARRAY[1..g_sJntNum] OF FB_PID;
	
	// rising edge generator for instrument information reading
	m_ReadLDP:R_TRIG;
	
	// code execute time measure
	m_codeTime : Profiler;
	
END_VAR

PROPERTY adjustFallEdge : BOOL
GET
adjustFallEdge := m_adjustFallEdge;
END_GET
END_PROPERTY

PROPERTY adjustOn : bool
GET
adjustOn := m_adjustOnFlag;
END_GET
END_PROPERTY

PROPERTY armIdx : int
GET
armIdx:=m_armIdx;
END_GET
END_PROPERTY

METHOD PROTECTED calcJaco : BOOL
VAR_IN_OUT CONSTANT
	i_DHJntPos :Vec6d;
END_VAR
VAR_IN_OUT
	r_jaco :Mat6d;
END_VAR
VAR_INPUT
END_VAR

VAR
	d1, L, a, b :LREAL;
	q3:LREAL;

	c1,c2,c4,c5,c6,c7 :LREAL;
	s1,s2,s4,s5,s6,s7 :LREAL;

END_VAR
d1:=GVL_SlaveArmKinematic.g_d1;
L:=m_instrument.instruTypeInfo.m_rodLength;
a:=m_instrument.instruTypeInfo.m_headLength;
//b:=m_instrument.instruTypeInfo.m_fingerLength;
b:=0;

q3:=i_DHJntPos[3];
c1:=COS(i_DHJntPos[1]);
c2:=COS(i_DHJntPos[2]);
c4:=COS(i_DHJntPos[4]);
c5:=COS(i_DHJntPos[5]);
c6:=COS(i_DHJntPos[6]);

s1:=SIN(i_DHJntPos[1]);
s2:=SIN(i_DHJntPos[2]);
s4:=SIN(i_DHJntPos[4]);
s5:=SIN(i_DHJntPos[5]);
s6:=SIN(i_DHJntPos[6]);

// jacobian with DH joints
r_jaco[1,1]:=b*(c6*(c5*(c1*s4 - c2*c4*s1) + s1*s2*s5) - s6*(c1*c4 + c2*s1*s4)) + a*(c5*(c1*s4 - c2*c4*s1) + s1*s2*s5) - L*s1*s2 + q3*s1*s2;
r_jaco[1,2]:=-c1*(a*(c2*s5 + c4*c5*s2) - L*c2 + q3*c2 + b*(c6*(c2*s5 + c4*c5*s2) + s2*s4*s6));
r_jaco[1,3]:=-c1*s2;
r_jaco[1,4]:=s1*s2*(a*(c2*s5 + c4*c5*s2) + b*(c6*(c2*s5 + c4*c5*s2) + s2*s4*s6)) - c2*(b*(c6*(c5*(c1*s4 - c2*c4*s1) + s1*s2*s5) - s6*(c1*c4 + c2*s1*s4)) + a*(c5*(c1*s4 - c2*c4*s1) + s1*s2*s5));
r_jaco[1,5]:=- (a*(c2*s5 + c4*c5*s2) + b*(c6*(c2*s5 + c4*c5*s2) + s2*s4*s6))*(c1*c4 + c2*s1*s4) - s2*s4*(b*(c6*(c5*(c1*s4 - c2*c4*s1) + s1*s2*s5) - s6*(c1*c4 + c2*s1*s4)) + a*(c5*(c1*s4 - c2*c4*s1) + s1*s2*s5));
r_jaco[1,6]:= b*(c6*(c5*(c1*s4 - c2*c4*s1) + s1*s2*s5) - s6*(c1*c4 + c2*s1*s4))*(c2*c5 - c4*s2*s5) + b*(s5*(c1*s4 - c2*c4*s1) - c5*s1*s2)*(c6*(c2*s5 + c4*c5*s2) + s2*s4*s6);


r_jaco[2,1]:=0;
r_jaco[2,2]:=c1*(a*(c5*(s1*s4 + c1*c2*c4) - c1*s2*s5) + b*(c6*(c5*(s1*s4 + c1*c2*c4) - c1*s2*s5) - s6*(c4*s1 - c1*c2*s4)) + L*c1*s2 - q3*c1*s2) - s1*(b*(c6*(c5*(c1*s4 - c2*c4*s1) + s1*s2*s5) - s6*(c1*c4 + c2*s1*s4)) + a*(c5*(c1*s4 - c2*c4*s1) + s1*s2*s5) - L*s1*s2 + q3*s1*s2);
r_jaco[2,3]:= c2;
r_jaco[2,4]:=- s1*s2*(a*(c5*(s1*s4 + c1*c2*c4) - c1*s2*s5) + b*(c6*(c5*(s1*s4 + c1*c2*c4) - c1*s2*s5) - s6*(c4*s1 - c1*c2*s4))) - c1*s2*(b*(c6*(c5*(c1*s4 - c2*c4*s1) + s1*s2*s5) - s6*(c1*c4 + c2*s1*s4)) + a*(c5*(c1*s4 - c2*c4*s1) + s1*s2*s5));
r_jaco[2,5]:=(a*(c5*(s1*s4 + c1*c2*c4) - c1*s2*s5) + b*(c6*(c5*(s1*s4 + c1*c2*c4) - c1*s2*s5) - s6*(c4*s1 - c1*c2*s4)))*(c1*c4 + c2*s1*s4) - (b*(c6*(c5*(c1*s4 - c2*c4*s1) + s1*s2*s5) - s6*(c1*c4 + c2*s1*s4)) + a*(c5*(c1*s4 - c2*c4*s1) + s1*s2*s5))*(c4*s1 - c1*c2*s4);
r_jaco[2,6]:=b*(c6*(c5*(c1*s4 - c2*c4*s1) + s1*s2*s5) - s6*(c1*c4 + c2*s1*s4))*(s5*(s1*s4 + c1*c2*c4) + c1*c5*s2) - b*(s5*(c1*s4 - c2*c4*s1) - c5*s1*s2)*(c6*(c5*(s1*s4 + c1*c2*c4) - c1*s2*s5) - s6*(c4*s1 - c1*c2*s4));

r_jaco[3,1]:=a*(c5*(s1*s4 + c1*c2*c4) - c1*s2*s5) + b*(c6*(c5*(s1*s4 + c1*c2*c4) - c1*s2*s5) - s6*(c4*s1 - c1*c2*s4)) + L*c1*s2 - q3*c1*s2;
r_jaco[3,2]:=-s1*(a*(c2*s5 + c4*c5*s2) - L*c2 + q3*c2 + b*(c6*(c2*s5 + c4*c5*s2) + s2*s4*s6));
r_jaco[3,3]:=-s1*s2;
r_jaco[3,4]:=- c2*(a*(c5*(s1*s4 + c1*c2*c4) - c1*s2*s5) + b*(c6*(c5*(s1*s4 + c1*c2*c4) - c1*s2*s5) - s6*(c4*s1 - c1*c2*s4))) - c1*s2*(a*(c2*s5 + c4*c5*s2) + b*(c6*(c2*s5 + c4*c5*s2) + s2*s4*s6));
r_jaco[3,5]:=- (a*(c2*s5 + c4*c5*s2) + b*(c6*(c2*s5 + c4*c5*s2) + s2*s4*s6))*(c4*s1 - c1*c2*s4) - s2*s4*(a*(c5*(s1*s4 + c1*c2*c4) - c1*s2*s5) + b*(c6*(c5*(s1*s4 + c1*c2*c4) - c1*s2*s5) - s6*(c4*s1 - c1*c2*s4)));
r_jaco[3,6]:=b*(c6*(c5*(s1*s4 + c1*c2*c4) - c1*s2*s5) - s6*(c4*s1 - c1*c2*s4))*(c2*c5 - c4*s2*s5) + b*(c6*(c2*s5 + c4*c5*s2) + s2*s4*s6)*(s5*(s1*s4 + c1*c2*c4) + c1*c5*s2);

r_jaco[4,1]:=0;
r_jaco[4,2]:=-s1;
r_jaco[4,3]:=0;
r_jaco[4,4]:=-c1*s2;
r_jaco[4,5]:=c1*c2*s4 - c4*s1;
r_jaco[4,6]:=s5*(s1*s4 + c1*c2*c4) + c1*c5*s2;

r_jaco[5,1]:=-1;
r_jaco[5,2]:=0;
r_jaco[5,3]:=0;
r_jaco[5,4]:=c2;
r_jaco[5,5]:=s2*s4;
r_jaco[5,6]:=c4*s2*s5 - c2*c5;

r_jaco[6,1]:=0;
r_jaco[6,2]:=c1;
r_jaco[6,3]:=0;
r_jaco[6,4]:=-s1*s2;
r_jaco[6,5]:=c1*c4 + c2*s1*s4;
r_jaco[6,6]:=c5*s1*s2 - s5*(c1*s4 - c2*c4*s1);
END_METHOD

METHOD PROTECTED checkIO : BOOL
VAR_INPUT
END_VAR

VAR
	startFlag:BOOL;
END_VAR
// check adjust button
m_adjustOnFlag := m_adjustDetect.run(m_adjustIO);
m_adjustFallEdgeDetect(CLK:=m_adjustOnFlag, Q=>m_adjustFallEdge);

// check trocar
m_trocarOnFlag := m_trocarDetect.run(m_adjustIO);

// check panel and instrument
m_panelOnFlag := m_panelDetect.run(m_panelInstrumentOnIO);
m_instruOnFlag := m_instruDetect.run(m_panelInstrumentOnIO);
m_instruNearFlag := m_instruNearDetect.run(m_panelInstrumentOnIO);

//read instrument information
IF FALSE = m_instruOnFlag THEN
	m_instrument.reset();
END_IF
m_ReadLDP(CLK:= m_instruOnFlag, Q=>startFlag );
// try to read again if instrument ID is undefined
startFlag := startFlag OR m_instrument.onChipData.m_ErrorID = 1;
m_instrument.readParameters(startFlag);


// check endoscope type and posture 
// only check when electric Knife is off 
IF SlaveArmControl.m_masterRobotData.m_electricKnifePedalTrigger[1] = 0 AND SlaveArmControl.m_masterRobotData.m_electricKnifePedalTrigger[2] = 0 THEN
	IF m_endoscopeTypeSwitch.check((m_panelInstrumentOnIO AND 16#20)=32) THEN
		IF m_instrument.curScopeType = EndoScopeType_30 THEN
			m_instrument.nextScopeType := EndoscopeType_0;
		ELSE
			m_instrument.nextScopeType := EndoscopeType_30;
		END_IF
	END_IF
	IF m_endoscopePostureSwitch.check((m_panelInstrumentOnIO AND 16#10)=16) AND m_instrument.curScopeType = EndoScopeType_30  THEN
		IF m_instrument.curScopePosture = EndoScopePosture_HeadDown THEN
			m_instrument.nextScopePosture := EndoscopePosture_HeadUp;
		ELSE
			m_instrument.nextScopePosture := EndoScopePosture_HeadDown;
		END_IF
	END_IF
END_IF
END_METHOD

PROPERTY cmdCartPose : REFERENCE TO ST_Frame
GET
cmdCartPose REF= m_cmdCartPose;
END_GET
END_PROPERTY

PROPERTY cmdCartTwist : REFERENCE to Vec6d
GET
cmdCartTwist REF= m_cmdCartTwist;
END_GET
END_PROPERTY

PROPERTY cmdJntCurrent : REFERENCE TO  Vec8d
GET
cmdJntCurrent ref= m_cmdJntCurrent;
END_GET
END_PROPERTY

PROPERTY cmdJntPos : REFERENCE TO Vec8d
GET
cmdJntPos REF= m_cmdJntPos;
END_GET
END_PROPERTY

PROPERTY cmdJntTrq :REFERENCE TO Vec8d
GET
cmdJntTrq REF= m_cmdJntTrq;
END_GET
END_PROPERTY

PROPERTY cmdJntVel : REFERENCE TO Vec8d
GET
cmdJntVel REF= m_cmdJntVel;
END_GET
END_PROPERTY

PROPERTY curCartPose : REFERENCE TO ST_Frame
GET
curCartPose ref=m_curCartPose;
END_GET
END_PROPERTY

PROPERTY curCartTwist : REFERENCE TO Vec6d
GET
curCartTwist ref=m_curCartTwist;
END_GET
END_PROPERTY

PROPERTY curDHJntPos :REFERENCE TO Vec6d
GET
curDHJntPos ref= m_curDHJntPos;
END_GET
END_PROPERTY

PROPERTY curDHJntVel :REFERENCE TO Vec6d
GET
curDHJntVel REF= m_curDHJntVel;
END_GET
END_PROPERTY

PROPERTY curGripAngle : LREAL
GET
curGripAngle:=m_curGripAngle;
END_GET
END_PROPERTY

PROPERTY curJntPos : REFERENCE TO Vec8d
GET
curJntPos ref=m_curJntPos;
END_GET
END_PROPERTY

PROPERTY curJntTrq : REFERENCE TO Vec8d
GET
curJntTrq ref=m_curJntTrq;
END_GET
END_PROPERTY

PROPERTY curJntVel :REFERENCE TO Vec8d
GET
curJntVel ref=m_curJntVel;
END_GET
END_PROPERTY

PROPERTY curLinkPos :REFERENCE TO Vec8d
GET
curLinkPos ref=m_curLinkPos;
END_GET
END_PROPERTY

PROPERTY curMotorPos : REFERENCE TO  Vec8d
GET
curMotorPos ref=m_curMotorPos;
END_GET
END_PROPERTY

METHOD PUBLIC enable : BOOL
VAR_IN_OUT CONSTANT
	i_jntIdx :Vec8i;
END_VAR
VAR
	i :INT ;
END_VAR
FOR i:=1 TO g_sJntNum DO
	IF 1= i_jntIdx[i] THEN
		m_joints[i].enable();
	ELSE
		m_joints[i].disable();
	END_IF
END_FOR
END_METHOD

PROPERTY filtJntCurrent :REFERENCE TO Vec8d
GET
filtJntCurrent ref= m_filtJntCurrent;
END_GET
END_PROPERTY

// from active joint position to cartesian pose in arm origin
METHOD PROTECTED forwardKinematic : BOOL
VAR_IN_OUT CONSTANT
	i_DHJntPos :Vec6d;
END_VAR
VAR_IN_OUT
	r_cartPose :ST_Frame;
END_VAR
VAR
	d1, L, a, b :LREAL;
	q3 :LREAL;

	c1,c2,c4,c5,c6,c7 :LREAL;
	s1,s2,s4,s5,s6,s7 :LREAL;
	DHRot :Mat3d;
	
	tmpRot1,tmpRot2 : Mat3d;

END_VAR
d1:=GVL_SlaveArmKinematic.g_d1;
L:=m_instrument.instruTypeInfo.m_rodLength;
a:=m_instrument.instruTypeInfo.m_headLength;
//b:=m_instrument.instruTypeInfo.m_fingerLength;
b:=0;

q3:=i_DHJntPos[3];
c1:=COS(i_DHJntPos[1]);
c2:=COS(i_DHJntPos[2]);
c4:=COS(i_DHJntPos[4]);
c5:=COS(i_DHJntPos[5]);
c6:=COS(i_DHJntPos[6]);

s1:=SIN(i_DHJntPos[1]);
s2:=SIN(i_DHJntPos[2]);
s4:=SIN(i_DHJntPos[4]);
s5:=SIN(i_DHJntPos[5]);
s6:=SIN(i_DHJntPos[6]);


// cartesian pose frame
r_cartPose.m_pos[1]:=a*(c5*(s1*s4 + c1*c2*c4) - c1*s2*s5) + b*(c6*(c5*(s1*s4 + c1*c2*c4) - c1*s2*s5) - s6*(c4*s1 - c1*c2*s4)) + L*c1*s2 - q3*c1*s2;
r_cartPose.m_pos[2]:=a*(c2*s5 + c4*c5*s2) - d1 - L*c2 + q3*c2 + b*(c6*(c2*s5 + c4*c5*s2) + s2*s4*s6);
r_cartPose.m_pos[3]:=L*s1*s2 - a*(c5*(c1*s4 - c2*c4*s1) + s1*s2*s5) - b*(c6*(c5*(c1*s4 - c2*c4*s1) + s1*s2*s5) - s6*(c1*c4 + c2*s1*s4)) - q3*s1*s2;

DHRot[1,1]:= c6*(c5*(s1*s4 + c1*c2*c4) - c1*s2*s5) - s6*(c4*s1 - c1*c2*s4);
DHRot[2,1]:=c6*(c2*s5 + c4*c5*s2) + s2*s4*s6;
DHRot[3,1]:=s6*(c1*c4 + c2*s1*s4) - c6*(c5*(c1*s4 - c2*c4*s1) + s1*s2*s5);

DHRot[1,2]:=- s6*(c5*(s1*s4 + c1*c2*c4) - c1*s2*s5) - c6*(c4*s1 - c1*c2*s4);
DHRot[2,2]:=c6*s2*s4 - s6*(c2*s5 + c4*c5*s2);
DHRot[3,2]:=s6*(c5*(c1*s4 - c2*c4*s1) + s1*s2*s5) + c6*(c1*c4 + c2*s1*s4);

DHRot[1,3]:= s5*(s1*s4 + c1*c2*c4) + c1*c5*s2;
DHRot[2,3]:= c4*s2*s5 - c2*c5;
DHRot[3,3]:=c5*s1*s2 - s5*(c1*s4 - c2*c4*s1);

// convert to tcp rotation
matMultiply(DHRot, GVL_SlaveArmKinematic.g_tcpRotation, r_cartPOSE.m_rot);

//TODO: need verify
// rotate tcp coordinate 180 degree about z axis if instrument is a head-up 30deg endoscope
IF m_instrument.instruType = InstruType_Endoscope AND m_instrument.curScopeType = EndoScopeType_30 AND m_instrument.curScopePosture = EndoscopePosture_HeadUp THEN
	tmpRot2 := rotZ(pi);
	tmpRot1 := r_cartPOSE.m_rot;
	matMultiply(tmpRot1, tmpRot2, r_cartPOSE.m_rot);
END_IF
END_METHOD

METHOD PUBLIC init : BOOL
VAR_INPUT
	i_armIdx:INT;
END_VAR
VAR 
	i :INT ;
	currentRatioMotor2Jnt: LREAL;
END_VAR
// arm statues init
m_armIdx:=i_armIdx;
m_curGripAngle:=0;
m_simGripAngle:=0;
m_instruJntBacklash := g_zeroVec5d;

// joint init
FOR i:=1 TO g_sJntNum DO
	IF i<4 THEN
		m_joints[i].init(m_armIdx, i,g_slaveArmCtrlCycleTime, 1);
	ELSE
		m_joints[i].init(m_armIdx, i,g_slaveArmCtrlCycleTime, 4);
	END_IF
END_FOR

// init joint encoder and position calculation
initJntPos();

// joint controller init
FOR i:=1 TO g_sJntNum DO 
	currentRatioMotor2Jnt:=GVL_SlaveMotorParameters.g_motorTrqConst[i]*GVL_SlaveMotorParameters.g_motorReduction[i]/1000;
	m_jntPIDCtrl[i].init(g_slaveArmCtrlCycleTime,GVL_slaveControlParameters.g_posKp[i],GVL_slaveControlParameters.g_posKd[i],
		GVL_slaveControlParameters.g_posKi[i], GVL_slaveControlParameters.g_posKiLimit[i]* currentRatioMotor2Jnt,
		GVL_slaveControlParameters.g_posCtrlLimit[i]*currentRatioMotor2Jnt);
END_FOR

// instrument init
m_instrument.init(i_armIdx);

// endosocpe toggle button check
m_endoscopeTypeSwitch.init(0, 500);
m_endoscopePostureSwitch.init(0,500);
END_METHOD

METHOD PUBLIC initJntPos : BOOL
VAR_INPUT
END_VAR
VAR
	i:INT ;
END_VAR
// joint init
FOR i:=1 TO g_sJntNum DO
	m_joints[i].initJntPos();
END_FOR

// update arm status if joint position is re-init
updateStatus();
END_METHOD

PROPERTY instruJntBacklash :REFERENCE TO Vec5d
GET
instruJntBacklash ref=m_instruJntBacklash;
END_GET
SET
m_instruJntBacklash := instruJntBacklash;
END_SET
END_PROPERTY

PROPERTY instrument : REFERENCE TO FB_Instrument
GET
instrument REF=m_instrument;
END_GET
END_PROPERTY

PROPERTY instruNear : BOOL
GET
instruNear := m_instruNearFlag;
END_GET
END_PROPERTY

PROPERTY instruOn : bool
GET
instruOn:=m_instruOnFlag;
END_GET
END_PROPERTY

// check if instrument is in ready position(far enough from romote center) for following manipulation
METHOD PUBLIC instruReady : BOOL
VAR_INPUT
END_VAR

VAR
	// check buffer
	checkBuffer :LREAL := 0.005;
END_VAR
IF NOT(m_instrument.onChipData.m_InstruReadSucceed) THEN
	instruReady :=FALSE;
	RETURN;
END_IF

instruReady := m_curJntPos[3] < (m_instrument.instruTypeInfo.m_rodLength+m_instrument.instruTypeInfo.m_headLength
									+ m_instrument.instruTypeInfo.m_fingerLength - GVL_SlaveArmKinematic.g_minInstruRCDis+checkBuffer);
END_METHOD

METHOD PUBLIC isEnabled : BOOL
VAR_IN_OUT CONSTANT
	i_jntIdx :Vec8i;
END_VAR
VAR
	i :INT ;
END_VAR
isEnabled := TRUE;
FOR i:=1 TO g_sJntNum DO
	IF 1= i_jntIdx[i] THEN
		isEnabled :=  (m_joints[i].isEnabled() AND isEnabled);
	END_IF
END_FOR
END_METHOD

PROPERTY isSingurality : bool
GET
isSingurality:=m_isSingularity;
END_GET
END_PROPERTY

PROPERTY jaco :REFERENCE TO Mat6d
GET
jaco ref= m_jaco;
END_GET
END_PROPERTY

PROPERTY jntGravity :REFERENCE TO Vec8d
GET
jntGravity ref=m_jntGravity;
END_GET
END_PROPERTY

PROPERTY linkSingle : REFERENCE TO Vec8d
GET
linkSingle ref=m_curLinkSingle;
END_GET
END_PROPERTY

PROPERTY PUBLIC massMat :REFERENCE TO Mat3d
GET
massMat ref=m_jntMassMat;
END_GET
END_PROPERTY

METHOD PROTECTED modifyJaco : BOOL
VAR_IN_OUT CONSTANT
	i_DHJntPos :Vec6d;
END_VAR
VAR_IN_OUT
	r_jaco :Mat6d;
END_VAR

VAR CONSTANT
	// modify joint2/3 position to avoid jacobian singularity
	m_Jnt2PosThres :LREAL := -165 * g_deg2Rad;
	m_Jnt3PosThres :LREAL := -0.03;
END_VAR

VAR
	d1, L, a, b :LREAL;
	q2, q3:LREAL;

	c1,c2,c4,c5,c6,c7 :LREAL;
	s1,s2,s4,s5,s6,s7 :LREAL;
END_VAR
d1:=GVL_SlaveArmKinematic.g_d1;
L:=m_instrument.instruTypeInfo.m_rodLength;
a:=m_instrument.instruTypeInfo.m_headLength;
//b:=m_instrument.instruTypeInfo.m_fingerLength;
b:=0;

q2 := i_DHJntPos[2];
IF q2 < m_Jnt2PosThres THEN
	q2 := m_Jnt2PosThres;
END_IF

q3:=i_DHJntPos[3];
IF q3 - L > m_Jnt3PosThres THEN
	q3:= L + m_Jnt3PosThres;
END_IF

c1:=COS(i_DHJntPos[1]);
c2:=COS(q2);
c4:=COS(i_DHJntPos[4]);
c5:=COS(i_DHJntPos[5]);
c6:=COS(i_DHJntPos[6]);

s1:=SIN(i_DHJntPos[1]);
s2:=SIN(q2);
s4:=SIN(i_DHJntPos[4]);
s5:=SIN(i_DHJntPos[5]);
s6:=SIN(i_DHJntPos[6]);

// jacobian with DH joints
r_jaco[1,1]:=b*(c6*(c5*(c1*s4 - c2*c4*s1) + s1*s2*s5) - s6*(c1*c4 + c2*s1*s4)) + a*(c5*(c1*s4 - c2*c4*s1) + s1*s2*s5) - L*s1*s2 + q3*s1*s2;
r_jaco[1,2]:=-c1*(a*(c2*s5 + c4*c5*s2) - L*c2 + q3*c2 + b*(c6*(c2*s5 + c4*c5*s2) + s2*s4*s6));
r_jaco[1,3]:=-c1*s2;
r_jaco[1,4]:=s1*s2*(a*(c2*s5 + c4*c5*s2) + b*(c6*(c2*s5 + c4*c5*s2) + s2*s4*s6)) - c2*(b*(c6*(c5*(c1*s4 - c2*c4*s1) + s1*s2*s5) - s6*(c1*c4 + c2*s1*s4)) + a*(c5*(c1*s4 - c2*c4*s1) + s1*s2*s5));
r_jaco[1,5]:=- (a*(c2*s5 + c4*c5*s2) + b*(c6*(c2*s5 + c4*c5*s2) + s2*s4*s6))*(c1*c4 + c2*s1*s4) - s2*s4*(b*(c6*(c5*(c1*s4 - c2*c4*s1) + s1*s2*s5) - s6*(c1*c4 + c2*s1*s4)) + a*(c5*(c1*s4 - c2*c4*s1) + s1*s2*s5));
r_jaco[1,6]:= b*(c6*(c5*(c1*s4 - c2*c4*s1) + s1*s2*s5) - s6*(c1*c4 + c2*s1*s4))*(c2*c5 - c4*s2*s5) + b*(s5*(c1*s4 - c2*c4*s1) - c5*s1*s2)*(c6*(c2*s5 + c4*c5*s2) + s2*s4*s6);


r_jaco[2,1]:=0;
r_jaco[2,2]:=c1*(a*(c5*(s1*s4 + c1*c2*c4) - c1*s2*s5) + b*(c6*(c5*(s1*s4 + c1*c2*c4) - c1*s2*s5) - s6*(c4*s1 - c1*c2*s4)) + L*c1*s2 - q3*c1*s2) - s1*(b*(c6*(c5*(c1*s4 - c2*c4*s1) + s1*s2*s5) - s6*(c1*c4 + c2*s1*s4)) + a*(c5*(c1*s4 - c2*c4*s1) + s1*s2*s5) - L*s1*s2 + q3*s1*s2);
r_jaco[2,3]:= c2;
r_jaco[2,4]:=- s1*s2*(a*(c5*(s1*s4 + c1*c2*c4) - c1*s2*s5) + b*(c6*(c5*(s1*s4 + c1*c2*c4) - c1*s2*s5) - s6*(c4*s1 - c1*c2*s4))) - c1*s2*(b*(c6*(c5*(c1*s4 - c2*c4*s1) + s1*s2*s5) - s6*(c1*c4 + c2*s1*s4)) + a*(c5*(c1*s4 - c2*c4*s1) + s1*s2*s5));
r_jaco[2,5]:=(a*(c5*(s1*s4 + c1*c2*c4) - c1*s2*s5) + b*(c6*(c5*(s1*s4 + c1*c2*c4) - c1*s2*s5) - s6*(c4*s1 - c1*c2*s4)))*(c1*c4 + c2*s1*s4) - (b*(c6*(c5*(c1*s4 - c2*c4*s1) + s1*s2*s5) - s6*(c1*c4 + c2*s1*s4)) + a*(c5*(c1*s4 - c2*c4*s1) + s1*s2*s5))*(c4*s1 - c1*c2*s4);
r_jaco[2,6]:=b*(c6*(c5*(c1*s4 - c2*c4*s1) + s1*s2*s5) - s6*(c1*c4 + c2*s1*s4))*(s5*(s1*s4 + c1*c2*c4) + c1*c5*s2) - b*(s5*(c1*s4 - c2*c4*s1) - c5*s1*s2)*(c6*(c5*(s1*s4 + c1*c2*c4) - c1*s2*s5) - s6*(c4*s1 - c1*c2*s4));

r_jaco[3,1]:=a*(c5*(s1*s4 + c1*c2*c4) - c1*s2*s5) + b*(c6*(c5*(s1*s4 + c1*c2*c4) - c1*s2*s5) - s6*(c4*s1 - c1*c2*s4)) + L*c1*s2 - q3*c1*s2;
r_jaco[3,2]:=-s1*(a*(c2*s5 + c4*c5*s2) - L*c2 + q3*c2 + b*(c6*(c2*s5 + c4*c5*s2) + s2*s4*s6));
r_jaco[3,3]:=-s1*s2;
r_jaco[3,4]:=- c2*(a*(c5*(s1*s4 + c1*c2*c4) - c1*s2*s5) + b*(c6*(c5*(s1*s4 + c1*c2*c4) - c1*s2*s5) - s6*(c4*s1 - c1*c2*s4))) - c1*s2*(a*(c2*s5 + c4*c5*s2) + b*(c6*(c2*s5 + c4*c5*s2) + s2*s4*s6));
r_jaco[3,5]:=- (a*(c2*s5 + c4*c5*s2) + b*(c6*(c2*s5 + c4*c5*s2) + s2*s4*s6))*(c4*s1 - c1*c2*s4) - s2*s4*(a*(c5*(s1*s4 + c1*c2*c4) - c1*s2*s5) + b*(c6*(c5*(s1*s4 + c1*c2*c4) - c1*s2*s5) - s6*(c4*s1 - c1*c2*s4)));
r_jaco[3,6]:=b*(c6*(c5*(s1*s4 + c1*c2*c4) - c1*s2*s5) - s6*(c4*s1 - c1*c2*s4))*(c2*c5 - c4*s2*s5) + b*(c6*(c2*s5 + c4*c5*s2) + s2*s4*s6)*(s5*(s1*s4 + c1*c2*c4) + c1*c5*s2);

r_jaco[4,1]:=0;
r_jaco[4,2]:=-s1;
r_jaco[4,3]:=0;
r_jaco[4,4]:=-c1*s2;
r_jaco[4,5]:=c1*c2*s4 - c4*s1;
r_jaco[4,6]:=s5*(s1*s4 + c1*c2*c4) + c1*c5*s2;

r_jaco[5,1]:=-1;
r_jaco[5,2]:=0;
r_jaco[5,3]:=0;
r_jaco[5,4]:=c2;
r_jaco[5,5]:=s2*s4;
r_jaco[5,6]:=c4*s2*s5 - c2*c5;

r_jaco[6,1]:=0;
r_jaco[6,2]:=c1;
r_jaco[6,3]:=0;
r_jaco[6,4]:=-s1*s2;
r_jaco[6,5]:=c1*c4 + c2*s1*s4;
r_jaco[6,6]:=c5*s1*s2 - s5*(c1*s4 - c2*c4*s1);
END_METHOD

PROPERTY panelOn : bool
GET
panelOn :=m_panelOnFlag;
END_GET
END_PROPERTY

PROPERTY rawJntCurrent :REFERENCE TO Vec8d
GET
rawJntCurrent ref=m_rawJntCurrent;
END_GET
END_PROPERTY

// check if instrument is in ready position(far enough from romote center) for following manipulation
METHOD PUBLIC readyForInstruMount : BOOL
VAR_INPUT
END_VAR

VAR
	// check buffer
	checkBuffer :LREAL := 0.01;
	i:INT;
END_VAR
readyForInstruMount := (m_curJntPos[3]> GVL_SlaveMotorParameters.g_maxDHJntPos[3]-checkBuffer AND m_panelOnFlag);

// make sure instrument joint at zero position
FOR i:=4 TO 8 DO
	IF m_curLinkSingle[i]>1*g_deg2rad AND m_curLinkSingle[i]< g_2pi - 1*g_deg2rad THEN
		readyForInstruMount:=FALSE;
		EXIT;
	END_IF
END_FOR
END_METHOD

METHOD PUBLIC resetInstruDepth : BOOL
VAR_INPUT
END_VAR
m_instruInvasionDepth :=GVL_SlaveMotorParameters.g_maxJntPos[3];
END_METHOD

METHOD PUBLIC setInstruDepth : BOOL
VAR_INPUT
END_VAR
m_instruInvasionDepth := m_curJntPos[3]-m_instrument.instruTypeInfo.m_rodLength -
			COS(m_curDHJntPos[5]+pi/2) *( m_instrument.instruTypeInfo.m_headLength + m_instrument.instruTypeInfo.m_fingerLength * COS(m_curDHJntPos[6]));
END_METHOD

PROPERTY simCartPose :REFERENCE TO ST_Frame
GET
simCartPose ref=m_simCartPose;
END_GET
END_PROPERTY

PROPERTY simDHJntPos :REFERENCE TO Vec6d
GET
simDHJntPos ref= m_simDHJntPos;
END_GET
END_PROPERTY

PROPERTY simGripAngle : LREAL
GET
simGripAngle:=m_simGripAngle;
END_GET
END_PROPERTY

PROPERTY simJaco :REFERENCE TO mat6d
GET
simJaco ref=m_simJaco;
END_GET
END_PROPERTY

PROPERTY simJacoInv :REFERENCE TO Mat6d
GET
simJacoInv ref= m_simJacoInv;
END_GET
END_PROPERTY

PROPERTY PUBLIC trocarOn : bool
GET
trocarOn := m_trocarOnFlag;
END_GET
END_PROPERTY

// update joints control command
METHOD PUBLIC updateCmds : BOOL
VAR_IN_OUT CONSTANT
	i_armCtrlCmd : ST_SlaveArmCtrlCmds;
END_VAR
VAR
	i:INT;
END_VAR
m_cmdJntTrq:=i_armCtrlCmd.m_cmdJntTrq;
m_cmdJntPos :=i_armCtrlCmd.m_cmdJntPos;
m_cmdJntVel :=i_armCtrlCmd.m_cmdJntVel;
m_cmdCartTwist := i_armCtrlCmd.m_cmdCartTwist;
m_cmdCartPose :=i_armCtrlCmd.m_cmdCartPose;
m_simJntPos:=i_armCtrlCmd.m_simJntPos;

// update simulated master arm
updateSimStatus();

// enable/disable joints
enable(i_armCtrlCmd.m_jntEnableFlag);

m_codeTime(START:=TRUE, RESET:=TRUE);
// position/torque control
FOR i:=1 TO g_sJntNum DO 
	IF i_armCtrlCmd.m_jntOPMode[i]=DriverOPMode_PosTrq THEN
		// position controller and gravity feedforward
		m_cmdJntTrq[i]:=m_jntPIDCtrl[i].run(m_cmdJntPos[i],m_curJntPos[i],m_cmdJntVel[i],m_curJntVel[i]);
		m_cmdJntTrq[i]:=m_cmdJntTrq[i]+m_jntGravity[i] + i_armCtrlCmd.m_FFJntTrq[i];
		m_joints[i].updateCmds(DriverOPMode_Trq,m_cmdJntPos[i],m_cmdJntTrq[i]);
	ELSIF i_armCtrlCmd.m_jntOPMode[i]=DriverOPMode_Trq THEN
		// gravity feedforward
		m_jntPIDCtrl[i].reset();
		m_cmdJntTrq[i]:=m_cmdJntTrq[i]+m_jntGravity[i];
		m_joints[i].updateCmds(DriverOPMode_Trq,m_cmdJntPos[i],m_cmdJntTrq[i]);
	ELSE
		m_jntPIDCtrl[i].reset();
		m_cmdJntTrq[i]:=0;
		IF i>3 THEN
			// add instrument joint backlash
			m_joints[i].updateCmds(DriverOPMode_Pos,m_cmdJntPos[i]+m_instruJntBacklash[i-3],m_cmdJntTrq[i]);
		ELSE
			m_joints[i].updateCmds(DriverOPMode_Pos,m_cmdJntPos[i],m_cmdJntTrq[i]);
		END_IF
	END_IF
	
END_FOR
m_codeTime(START:=FALSE);
END_METHOD

METHOD PUBLIC updateDyna : BOOL
VAR_IN_out constant
	slaveDynaData : ST_SlaveDynaData;
END_VAR
m_jntMassMat:=slaveDynaData.m_massMat[m_armIdx];
m_jntGravity[1]:=slaveDynaData.m_gravity[m_armIdx][1];
m_jntGravity[2]:=slaveDynaData.m_gravity[m_armIdx][2];
m_jntGravity[3]:=slaveDynaData.m_gravity[m_armIdx][3];
END_METHOD

METHOD PUBLIC updateSimStatus : BOOL
VAR_INPUT
END_VAR
// instrument kinematic
m_instrument.instruFK(m_simJntPos, m_simDHJntPos, m_simGripAngle);

// simulated cartesion pose 
forwardKinematic(m_simDHJntPos,m_simCartPose);

// simulated jacobian
modifyJaco(m_simDHJntPos,m_simJaco);
m_isSingularity:=NOT(invMat6(m_simJaco, m_simJacoInv));
END_METHOD

// update arm status, including kinematic and dynamic
METHOD PUBLIC updateStatus : BOOL
VAR_INPUT
END_VAR
VAR 
	i,j:INT;
END_VAR
// update joint data
FOR i:=1 TO g_sJntNum DO
	m_joints[i].updateStatus();
END_FOR

// check IO informantion
checkIO();

// get joint data
FOR i:=1 TO g_sJntNum DO
	// remove instrument joint backlash
	IF i>3 THEN
		m_curMotorPos[i]:=m_joints[i].motorPos - m_instruJntBacklash[i-3];
		m_curLinkPos[i]:=m_joints[i].linkPos - m_instruJntBacklash[i-3];
		m_curLinkSingle[i]:=m_joints[i].linkSingle - m_instruJntBacklash[i-3];
		m_curJntPos[i]:=m_joints[i].jntPos - m_instruJntBacklash[i-3];
	ELSE
		m_curMotorPos[i]:=m_joints[i].motorPos;
		m_curLinkPos[i]:=m_joints[i].linkPos;
		m_curLinkSingle[i]:=m_joints[i].linkSingle;
		m_curJntPos[i]:=m_joints[i].jntPos;
	END_IF
	m_curJntVel[i]:=m_joints[i].jntVel;
	m_curJntTrq[i]:=m_joints[i].jntTrq;
	m_rawJntCurrent[i]:=m_joints[i].rawCurrent;
	m_filtJntCurrent[i]:=m_joints[i].filtCurrent;
	m_cmdJntCurrent[i]:=m_joints[i].cmdCurrent;
END_FOR 

// instrument kinematic
m_instrument.instruFK(m_curJntPos, m_curDHJntPos, m_curGripAngle);

// cartesion pose
forwardKinematic(m_curDHJntPos,m_curCartPose);

// jacobian
calcJaco(m_curDHJntPos,m_jaco);

// DH joint velocity
m_instrument.instruJntVelFK(m_curJntVel, m_curDHJntVel);

// cartesian twist
matMultiVec(m_jaco, m_curDHJntVel, m_curCartTwist);
END_METHOD

END_FUNCTION_BLOCK

// ---- FBs_Robots/FB_SlaveJoint.TcPOU
FUNCTION_BLOCK FB_SlaveJoint EXTENDS FB_JointBase
VAR_INPUT
END_VAR
VAR_OUTPUT
END_VAR
VAR
	// power box joint motor rated current
	m_wristJntRatedCurrent : DINT := 200;

END_VAR

METHOD PUBLIC init : BOOL
VAR_INPUT
	i_armIdx :INT;
	i_jntIdx :INT;
	i_controlCycleTime :LREAL;
	// velocity is calculated every (m_velCalcCycles) control cycles
	// TODO: insturment joint motor can not reach 4k now, so calculate their velocity with 1k frequency, need to remove later
	i_velCalcCycles :INT;
END_VAR
m_armIdx:=i_armIdx;
m_jntIdx:=i_jntIdx;
m_cycleTime := i_controlCycleTime;
m_velCalcCycles :=MAX(i_velCalcCycles,1);

// hardware parameters
m_motorEncoderRes :=GVL_SlaveMotorParameters.g_incEncoderRes[i_jntIdx];
m_linkEncoderRes :=GVL_SlaveMotorParameters.g_absEncoderRes[i_jntIdx];
m_motorReduction :=GVL_SlaveMotorParameters.g_motorReduction[i_jntIdx];
m_linkEncoderReduction :=GVL_SlaveMotorParameters.g_absEncoderReduction[i_jntIdx];
m_trqConst :=GVL_SlaveMotorParameters.g_motorTrqConst[i_jntIdx];
m_maxCurrent :=GVL_SlaveMotorParameters.g_motorMaxCurrent[i_jntIdx];
m_motorDir :=GVL_SlaveMotorParameters.g_motorDir[i_jntIdx];								
m_minJntPos	:=GVL_SlaveMotorParameters.g_minJntPos[i_jntIdx];
m_maxJntPos	:=GVL_SlaveMotorParameters.g_maxJntPos[i_jntIdx];

//link encoder calibartion data
m_linkEncoderDir :=GVL_SlaveJointEncoderCaliData.g_asbEncoderDir[i_jntIdx];
m_minLinkEncoder :=GVL_SlaveJointEncoderCaliData.g_minLinkEncoder[i_armIdx, i_jntIdx] - m_linkEncoderDir*GVL_SlaveJointEncoderCaliData.g_linkEncLimitBuffer; // expand limit
m_maxLinkEncoder :=GVL_SlaveJointEncoderCaliData.g_maxLinkEncoder[i_armIdx, i_jntIdx] + m_linkEncoderDir*GVL_SlaveJointEncoderCaliData.g_linkEncLimitBuffer; // expand limit
m_caliLinkEncoder :=GVL_SlaveJointEncoderCaliData.g_caliLinkEncoder[i_armIdx, i_jntIdx];
m_linkEncCaliJntPos :=GVL_SlaveJointEncoderCaliData.g_linkEncCaliJntPos[i_jntIdx];
m_linkEncZeroCross :=GVL_SlaveJointEncoderCaliData.g_linkEncZeroCross[i_armIdx, i_jntIdx];
m_multiCycles :=GVL_SlaveJointEncoderCaliData.g_multipleCyclesJoint[i_armIdx,i_jntIdx];

// convert cali link encoder if joint cross zero
IF 1=m_linkEncZeroCross THEN
	IF 1=m_linkEncoderDir AND m_caliLinkEncoder < m_minLinkEncoder THEN
		m_caliLinkEncoder := GVL_SlaveJointEncoderCaliData.g_caliLinkEncoder[i_armIdx, i_jntIdx] + m_linkEncoderRes;
	ELSIF -1=m_linkEncoderDir AND m_caliLinkEncoder < m_maxLinkEncoder THEN
		m_caliLinkEncoder := GVL_SlaveJointEncoderCaliData.g_caliLinkEncoder[i_armIdx, i_jntIdx] + m_linkEncoderRes;
	END_IF
END_IF

// macro data
m_trq2CurrentRatio:=m_motorDir * 1000.0/(m_trqConst*m_motorReduction);
m_current2TrqRatio:=m_motorDir * (m_trqConst*m_motorReduction)/1000.0;
m_linkEnc2PosRatio := 2*PI*m_linkEncoderDir/(m_linkEncoderReduction*m_linkEncoderRes);
m_motorEnc2PosRatio := 2*PI * m_motorDir/(m_motorReduction * m_motorEncoderRes);

// motor data init
m_rawJntVel :=0;
m_curJntVel:=0;
m_curJntTrq :=0;
m_rawCurrent :=0;
m_filtCurrent :=0;
m_cmdJntVel :=0.0;
m_cmdJntTrq :=0.0;
m_cmdCurrent := 0.0;

// filter init
m_jntVelLpf.init(1, GVL_SlaveControlParameters.g_curJntVelLpfCutoffFreq, g_slaveArmCtrlFreq/m_velCalcCycles);
m_cmdTrqLpf.init(1, GVL_SlaveControlParameters.g_cmdJntTrqLpfCutoffFreq, g_slaveArmCtrlFreq);
m_curTrqLpf.init(1, GVL_SlaveControlParameters.g_curJntTrqLpfCutoffFreq, g_slaveArmCtrlFreq);

// driver init value
m_motorOutputs.m_controlWord:=DriverCtrlWord_INIT;
m_motorOutputs.m_opMode:=INT_TO_SINT(DriverOPMode_Pos);
m_motorOutputs.m_cmdCurrent:=0;
m_motorOutputs.m_cmdMotorEncoder:=m_motorInputs.m_motorEncoder;
END_METHOD

METHOD PUBLIC updateCmds : BOOL
VAR_INPUT
	i_opMode : E_DriverOPMode;
	i_cmdPos :LREAL;
	i_cmdTrq :LREAL;
END_VAR
VAR
	filtCmdTrq :LREAL;
END_VAR
SUPER^.updateCmds(i_opMode, i_cmdPos, i_cmdTrq);

// write SDO data
writeSDOData();
END_METHOD

METHOD PROTECTED writeSDOData : BOOL
VAR_INPUT
END_VAR
VAR
	SDOSubIndexMode :WORD;
	SDOSubIndexCur :WORD;
END_VAR
//动力盒移动关节和器械旋转关节，共享一个控制字，由SDO写入
IF (m_jntIdx=3) OR (m_jntIdx=8)  THEN
	SDOSubIndexMode :=16#609B;
	SDOSubIndexCur:=16#6098;
//动力盒3、5号电机为一个驱动器，共享一个控制字，由SDO写入
ELSIF (m_jntIdx=4) OR (m_jntIdx=6)  THEN
	SDOSubIndexMode :=16#609C;
	SDOSubIndexCur:=16#6099;
//动力盒2、4号电机为一个驱动器，共享一个控制字，由SDO写入
ELSIF (m_jntIdx=5) OR (m_jntIdx=7)  THEN
	SDOSubIndexMode :=16#609D;
	SDOSubIndexCur:=16#609A;
END_IF

IF m_jntIdx <3 THEN
	RETURN;
END_IF

// write driver operation mode if it changs
IF  m_jntIdx >=3 AND m_jntIdx <=7 THEN
	m_opModeSDOWrite(sNetID:= GVL_SlaveJointEncoderCaliData.g_slaveArmNetID[m_armIdx],
					nSlaveAddr := GVL_SlaveJointEncoderCaliData.g_slaveJointNetPort[m_armIdx,m_jntIdx],
					nSubIndex:=0,nIndex:=SDOSubIndexMode,pSrcBuf:=ADR(m_motorOutputs.m_opMode),cbBufLen:=SIZEOF(m_motorOutputs.m_opMode),bExecute:=TRUE);
	IF NOT m_opModeSDOWrite.bBusy THEN
		m_opModeSDOWrite(bExecute:=FALSE);
	END_IF
END_IF

// write max motor current if it changes and works in position mode
IF m_jntIdx >=4 AND m_jntIdx <=8  THEN 
	m_MotorCurrentSDOWrite(sNetID:= GVL_SlaveJointEncoderCaliData.g_slaveArmNetID[m_armIdx],
					nSlaveAddr := GVL_SlaveJointEncoderCaliData.g_slaveJointNetPort[m_armIdx,m_jntIdx],
					nSubIndex:=0,nIndex:=SDOSubIndexCur,pSrcBuf:=ADR(m_wristJntRatedCurrent),cbBufLen:=SIZEOF(m_wristJntRatedCurrent),bExecute:=TRUE);
	IF NOT m_MotorCurrentSDOWrite.bBusy THEN
		m_MotorCurrentSDOWrite(bExecute:=FALSE);
	END_IF
END_IF
END_METHOD

END_FUNCTION_BLOCK

// ---- FBs_Auxiliary/FB_InstrumentDetect.TcPOU
FUNCTION_BLOCK FB_InstrumentDetect
VAR_INPUT
END_VAR
VAR_OUTPUT
END_VAR
VAR
	m_instruOnCounts :INT :=0;
	m_InstruOnCountThres :INT :=50;
END_VAR

// check if instrument is on
METHOD run : BOOL
VAR_INPUT
	IOValue :UDINT;
END_VAR
//Instrument single   At installation--2#0*0*   not installation --2#1*1*  And Hall single --2#100 0000
IF (IOValue AND 10#10) = 0  THEN
	m_instruOnCounts := MIN( m_instruOnCounts +1,m_InstruOnCountThres);
ELSIF (IOValue AND 10#10) = 10  THEN
	m_instruOnCounts :=0;
END_IF
run := m_instruOnCounts >= m_InstruOnCountThres;
END_METHOD

END_FUNCTION_BLOCK

// ---- FBs_Auxiliary/FB_InstruNearDetect.TcPOU
FUNCTION_BLOCK FB_InstruNearDetect
VAR_INPUT
END_VAR
VAR_OUTPUT
END_VAR
VAR
	m_instruNearCounts :INT :=0;
	m_InstruNearCountThres :INT :=50;
END_VAR

// check if instrument is near
METHOD run : BOOL
VAR_INPUT
	IOValue :UDINT;
END_VAR
//Instrument single   At installation--2#0*0*   not installation --2#1*1*  And Hall single --2#100 0000
IF (IOValue AND 10#64) = 64  THEN
	m_instruNearCounts := MIN( m_instruNearCounts +1,m_InstruNearCountThres);
ELSE
	m_instruNearCounts := 0;
END_IF

run := m_instruNearCounts >= m_InstruNearCountThres;
END_METHOD

END_FUNCTION_BLOCK

// ---- FBs_Auxiliary/FB_AdjustDetect.TcPOU
FUNCTION_BLOCK FB_AdjustDetect
VAR_INPUT
END_VAR
VAR_OUTPUT
END_VAR
VAR
	m_adjustOnCounts :INT :=0;
	m_adjustOnCountThres :INT :=50;
END_VAR

// check if instrument is on
METHOD run : BOOL
VAR_INPUT
	IOValue :UDINT;
END_VAR
// adjust io is 3th bit 
IF 8=(IOValue AND 10#8) THEN
	m_adjustOnCounts :=MIN(m_adjustOnCounts +1,m_adjustOnCountThres);
ELSE
	m_adjustOnCounts :=0;
END_IF

run := m_adjustOnCounts >= m_adjustOnCountThres;
END_METHOD

END_FUNCTION_BLOCK

// ---- FBs_Auxiliary/FB_IOToggleCheck.TcPOU
// return true if IO is triggerd for a set time period
// only return ture for one cycle, waiting for IO to be released and check for next time
FUNCTION_BLOCK FB_IOToggleCheck
VAR
	// IO type, 0- normally-opend IO; 1- normally-closed IO
	m_IOType :INT :=0;
	
	// counts after IO  is triggerd
	m_IOOnCounts :INT;
	
	// counts threshold indicating IO is trully triggerd
	m_IOOnCountThres :INT :=100;
END_VAR

METHOD check : BOOL
VAR_INPUT
	IOValue :BOOL;
END_VAR
check:=false;
IF (0=m_IOType and IOValue) OR (1=m_IOType AND NOT(IOValue)) THEN
	m_IOOnCounts := MIN(m_IOOnCounts +1, m_IOOnCountThres);
ELSE
	IF m_IOOnCounts>=m_IOOnCountThres THEN
		check:=TRUE;
	END_IF
	 m_IOOnCounts :=0;
END_IF
END_METHOD

METHOD init : BOOL
VAR_INPUT
	i_IOType :INT;
	i_triggerCounts:INT;
END_VAR
m_IOType:=i_IOType;
m_IOOnCountThres := i_triggerCounts;
END_METHOD

END_FUNCTION_BLOCK

// ---- FBs_Robots/FB_Instrument.TcPOU
FUNCTION_BLOCK FB_Instrument

VAR_IN_OUT CONSTANT
	i_slaveArm	:FB_SlaveArm;
END_VAR

VAR
	// instrument type
	m_instruType : 	E_InstrumentType := InstruType_UNKNOWM;
	
	// instrument type info
	m_instruTypeInfo : 	ST_InstruTypeInfo;
	
	//The state and parameters readed from the instrument
	m_onChipData:ST_InstruOnChipData;
	
	// current and max allowed read tries
	m_curReadTries :INT :=0;
	m_maxReadTries :INT := 2;
	
	//IP of operating arm
	m_armNetId:T_AmsNetId; 	
	
	//Joint port number
	m_jointInstruAddr:UINT;	
	
	//LED port address
	m_LEDAddr:UINT;		

	// joint position when instrument is at ZERO posture
	m_jntPosOffset:Vec8d;
	
	// instrument wrist DH joint limit
	m_wristMinDHJntPos :Vec3d;
	m_wristMaxDHJntPos :Vec3d;
	
	// reduction from motor joint to endoscope rotate joint
	m_endoscopeRotateReduction :LREAL := 2.0/3.0;
	
	// endoscope rotation joint index
	m_endoscopeRotJntIdx :INT :=8;
	
	//endoscope type
	m_curEndoscopeType :E_EndoscopeType:=EndoScopeType_30;
	m_nextEndoscopeType :E_EndoscopeType:=EndoScopeType_30;
	
	//endoscope posutre
	m_curEndoscopePosture :E_EndoscopePosture:=EndoscopePosture_HeadDown;
	m_nextEndoscopePosture :E_EndoscopePosture:=EndoscopePosture_HeadDown;
	
	// udint code for zero position
	m_zeroPosCode : UDINT;
	
	// joint4 zero position, which is supposed to be a contant value
	m_jnt4ZeroPos :LREAL := 5.7;
	
	//reset arm  LED flag
	m_resetArmLEDFlag : BOOL :=TRUE;
	
	// variables used to read instrument information
	m_Step:INT;
	m_Value:UDINT;
	m_ReadDelay:TON;
	m_DealyTime:TIME:=T#0.5S;
	m_IDReadResult:UDINT;
	m_IDResult:ULINT;
	m_SeriesReadResult:UDINT;
	m_PosReadResult:UDINT;
	m_PosL1,m_PosL2,m_PosL3:UDINT;
	m_signL1,m_signL2,m_signL3:UDINT;
	m_UsageReadResult:ULINT;
	m_InstruUsageToLED:ULINT;
	
	m_HaveRecord:BOOL;
	m_SdoWrite:FB_EcCoESdoWrite;
	m_SdoRead:FB_EcCoESdoRead;
	
	//variables used to read-write instrument number of use
	m_useNumStep : INT;
	m_ReadNumDelay:TON;
	m_useNumReadResult:ULINT;
	m_useNumSendToLED:ULINT;
	
	// rising edge generator for instrument information reading
	m_writeLDP:R_TRIG;
	
END_VAR

METHOD PROTECTED checkInstruType : BOOL
VAR_INPUT
END_VAR
VAR
	i:INT;
END_VAR
// search instrument type
checkInstruType :=FALSE;
FOR i:=1 TO g_instruTypeNum DO 
	IF g_instruTypePool[i].m_InstruID = m_onChipData.m_InstruID THEN
		checkInstruType:=TRUE;
		m_instruTypeInfo := g_instruTypePool[i];
		EXIT;
	END_IF
END_FOR

// return directly if instrument ID is invalid
IF NOT(checkInstruType) THEN
	RETURN;
END_IF
IF m_onChipData.m_InstruID = InstruType_NewEndoscope THEN
	m_instruType := InstruType_Endoscope;
	m_endoscopeRotateReduction := 1.0;
	m_endoscopeRotJntIdx := 7;
ELSE
	m_instruType := m_onChipData.m_InstruID;
	m_endoscopeRotateReduction := 2.0/3.0;
	m_endoscopeRotJntIdx := 8;
END_IF

// update DH joint limit
m_instruTypeInfo.m_rodLength := m_instruTypeInfo.m_rodLength - GVL_SlaveArmKinematic.g_panelHeight;
m_wristMinDHJntPos[1]:=-m_instruTypeInfo.m_rollLimit;
m_wristMaxDHJntPos[1]:=m_instruTypeInfo.m_rollLimit;
m_wristMinDHJntPos[2]:=-m_instruTypeInfo.m_pitchLimit-pi/2;
m_wristMaxDHJntPos[2]:=m_instruTypeInfo.m_pitchLimit-pi/2;
m_wristMinDHJntPos[3]:=-m_instruTypeInfo.m_yawLimit;
m_wristMaxDHJntPos[3]:=m_instruTypeInfo.m_yawLimit;
END_METHOD

PROPERTY curScopePosture : E_EndoscopePosture
GET
curScopePosture:= m_curEndoscopePosture;
END_GET
SET
m_curEndoscopePosture := curScopePosture;
END_SET
END_PROPERTY

PROPERTY curScopeType : E_EndoscopeType
GET
curScopeType := m_curEndoscopeType;
END_GET
SET
m_curEndoscopeType := curScopeType;
END_SET
END_PROPERTY

METHOD PUBLIC gripAngleMap : BOOL
VAR_INPUT
	// master gripper angle
	i_masterGripAng :LREAL;
END_VAR

VAR_OUTPUT
	// slave instrument gripper angle
	o_instruGripAngle :LREAL;
	
	// slave instrument grip force	
	o_instruGripForceLevel :LREAL;
END_VAR

VAR
	gripLevel :REAL;
END_VAR
// suppose finger is  closed and zero force if instrument has only one finger
IF m_instruTypeInfo.m_isSingleFinger THEN
	o_instruGripAngle := 0;
	o_instruGripForceLevel:= 0;
	RETURN;
END_IF 

// finger closed and force applied
IF i_masterGripAng < g_masterGripForceStartAng THEN
	o_instruGripAngle := g_minSlaveGripAngle;
	// NOTE: force is applied from 50%，as minimum gripper angle already apply some sort of force
	o_instruGripForceLevel := 50+50*(g_masterGripForceStartAng - i_masterGripAng)/(g_masterGripForceStartAng - g_minMasterGripAngle);
// finger open
ELSE
	o_instruGripAngle := (g_maxMasterGripAngle - i_masterGripAng)/(g_maxMasterGripAngle - g_masterGripForceStartAng);
	o_instruGripAngle :=m_instruTypeInfo.m_maxGripAngle - o_instruGripAngle * (m_instruTypeInfo.m_maxGripAngle - g_minSlaveGripAngle);
	o_instruGripAngle := LIMIT(g_minSlaveGripAngle, o_instruGripAngle, m_instruTypeInfo.m_maxGripAngle );
	o_instruGripForceLevel:=0;
END_IF
END_METHOD

METHOD PUBLIC init : BOOL
VAR_INPUT
	armIdx :INT;
END_VAR
VAR
	i:INT;
END_VAR
//Update the IP and port number of the operating arm
m_armNetId:=GVL_SlaveJointEncoderCaliData.g_slaveArmNetID[armIdx];
m_jointInstruAddr:=GVL_SlaveJointEncoderCaliData.g_slaveJointNetPort[armIdx,4];
m_LEDAddr := GVL_SlaveJointEncoderCaliData.g_slaveLEDNetPort[armIdx];

// init joint motion range
FOR i:=1 TO 3 DO
	m_wristMinDHJntPos[i]:=GVL_SlaveMotorParameters.g_minDHJntPos[i+3];
	m_wristMaxDHJntPos[i]:=GVL_SlaveMotorParameters.g_maxDHJntPos[i+3];
END_FOR
END_METHOD

METHOD PUBLIC initInstruJntPos : BOOL
VAR_INPUT
	m_curJntPos :Vec8d;
END_VAR

VAR
	i:INT;
END_VAR
FOR i := 4 TO 8 BY 1 DO
	m_jntPosOffset[i]:=m_curJntPos[i];
END_FOR
END_METHOD

// convert motor joint position to DH joint position
METHOD PUBLIC instruFK : BOOL
VAR_IN_OUT CONSTANT
	// motor joint position of slave arm
	i_jntPos :Vec8d;
END_VAR

VAR_IN_OUT
	// instrument DH  joint positon
	r_DHJntPos :Vec6d;

	// gripper angle
	r_gripAngle :LREAL;
END_VAR

VAR
	jntPosL1,jntPosL2,jntPosL3,jntPosL4,jntPosL5 :LREAL;
	gripAngle:LREAL;
	kx,ky,kz, k13, k23,openAngleDir:LREAL;
END_VAR
r_DHJntPos[1]:=i_jntPos[1];
r_DHJntPos[2]:=i_jntPos[2];
r_DHJntPos[3]:=i_jntPos[3];

// kinematic variables
openAngleDir:=-1;
kx:=-1;
ky:=m_instruTypeInfo.m_k2;
kz:=m_instruTypeInfo.m_k1;
k13:=m_instruTypeInfo.m_k3;
k23:=m_instruTypeInfo.m_k3;


// ################## endoscope ############################
IF m_instruType = InstruType_endoscope THEN
	r_DHJntPos[4]:=m_endoscopeRotateReduction*(i_jntPos[m_endoscopeRotJntIdx]-m_jntPosOffset[m_endoscopeRotJntIdx]);
	IF m_curEndoscopeType = EndoScopeType_30 THEN
		r_DHJntPos[5]:=-pi/2+30*g_deg2Rad;
	ELSE
		r_DHJntPos[5]:=-pi/2;
	END_IF
	r_DHJntPos[6]:=0;
	RETURN;
END_IF

// ################## ultrosonic knief ############################
IF m_instruType = InstruType_UltrasoundKnifeS OR m_instruType = InstruType_UltrasoundKnifeU THEN
	r_DHJntPos[4]:=-(i_jntPos[8]-m_jntPosOffset[8])/kx;
	r_DHJntPos[5]:=-pi/2;
	r_DHJntPos[6]:=0;
	r_gripAngle:=ultrasoundKnifeGripAngleFK(i_jntPos[6]-m_jntPosOffset[6]);
	RETURN;
END_IF


//#################### instrument forward kinematic ############
// convert motor joint position to instrument joint position
jntPosL1:=(i_jntPos[4]-m_jntPosOffset[4]);
jntPosL2:=(i_jntPos[5]-m_jntPosOffset[5]);
jntPosL3:=(i_jntPos[6]-m_jntPosOffset[6]);
jntPosL4:=-(i_jntPos[7]-m_jntPosOffset[7]);
jntPosL5:=-(i_jntPos[8]-m_jntPosOffset[8]);

// diable L1 if instrument is single finger
IF m_instruTypeInfo.m_isSingleFinger THEN
	jntPosL1 := -jntPosL2;
END_IF

// instrument FK in local coordinate
r_DHJntPos[4]:=jntPosL4/kx;
r_DHJntPos[5]:=jntPosL3/ky;
r_DHJntPos[6]:=(jntPosL1-jntPosL2-2*r_DHJntPos[5]*k13*kz)/(2*openAngleDir*kz);

// convert instrument rotation to arm DH joint position
r_DHJntPos[5]:=-r_DHJntPos[5]-pi/2;
r_DHJntPos[6]:=-r_DHJntPos[6];

// grip angle
gripAngle:=(jntPosL1+jntPosL2)/(openAngleDir*kz);

//################### gripper angle handle #################
IF (InstruType_ProGraspForceps=m_instruType OR InstruType_ForceBipolar=m_instruType) THEN//细齿无创抓钳
	proGrsapForcepsGripAngleFK(frontAngle:= gripAngle, endAngle=> r_gripAngle);

ELSIF (InstruType_CauteryHook = m_instruType OR InstruType_CauterySpatula = m_instruType) THEN//单级电钩
	r_gripAngle:=0;
ELSE
	r_gripAngle:=gripAngle;
END_IF
END_METHOD

METHOD PROTECTED InstruIDRecord :ARRAY [1..100] OF  ULINT
VAR_INPUT
	i_NewValue:ULINT;
	i_ArrayData:ARRAY [1..100] OF ULINT;
END_VAR

VAR
	k1:INT;
	Have_Data:BOOL;
END_VAR
FOR k1:= 1 TO 100 BY 1 DO
	IF i_NewValue=i_ArrayData[k1] THEN
		Have_Data:=TRUE;
		EXIT;
	ELSE
		Have_Data:=FALSE;
	END_IF
END_FOR

IF Have_Data=FALSE THEN
	FOR k1:= 1 TO 99 BY 1 DO
		InstruIDRecord[k1+1]:=i_ArrayData[k1];
	END_FOR
	InstruIDRecord[1]:=i_NewValue;
ELSE
	InstruIDRecord:=i_ArrayData ;
END_IF
END_METHOD

METHOD PUBLIC instruIK : BOOL
VAR_INPUT
	// DH  joint positon
	i_DHJntPos :Vec6d;

	// gripper angle
	i_gripAngle :LREAL;
	
END_VAR
VAR_OUTPUT
	o_jntPos:Vec8d;
END_VAR
VAR
	gripAngle:LREAL;
	i:INT;
	rot_x:lreal;
	rot_y:lreal;
	rot_z:lreal;

	kx,ky,kz,k13,k23:LREAL;
	d,ra:LREAL;
	
	m_gripAnglePbox:Vec8d;

END_VAR
o_jntPos[1] := i_DHJntPos[1];
o_jntPos[2] := i_DHJntPos[2];
o_jntPos[3] := i_DHJntPos[3];

// kinematic variables
d:=-1;
kx:=-1;
ky:=m_instruTypeInfo.m_k2;
kz:=m_instruTypeInfo.m_k1;
k13:=m_instruTypeInfo.m_k3;
k23:=m_instruTypeInfo.m_k3;

// ################## endoscope ############################
//IF m_instruType = InstruType_endoscope THEN
//	o_jntPos[8] := i_DHJntPos[4]/m_endoscopeRotateReduction + m_jntPosOffset[m_endoscopeRotJntIdx];
//	o_jntPos[4]:=0;
//	o_jntPos[5]:=0;
//	o_jntPos[6]:=0;
//	o_jntPos[7]:=0;
//	RETURN;
//END_IF

//################### gripper angle handle #################
IF (InstruType_ProGraspForceps=m_instruType OR InstruType_ForceBipolar=m_instruType) THEN//细齿无创抓钳
	proGrsapForcepsGripAngleIK(endAngle:= i_gripAngle, frontAngle=> gripAngle);
	
ELSIF (InstruType_CauteryHook = m_instruType OR InstruType_CauterySpatula = m_instruType)  THEN//单级电钩\电铲
	gripAngle:=0;
	
ELSE
	gripAngle:=i_gripAngle;
END_IF

// ################# instrument inverse kinematic ##############
// convert arm DH joint position to  instrument rotation
rot_x:=i_DHJntPos[4];
rot_y:=-i_DHJntPos[5]-pi/2;
rot_z:=-i_DHJntPos[6];

// ################## ultrosonic knief ############################
IF InstruType_UltrasoundKnifeS = onChipData.m_InstruID OR InstruType_UltrasoundKnifeU = onChipData.m_InstruID THEN
	m_gripAnglePbox[4]:=0;
	m_gripAnglePbox[5]:=0;
	m_gripAnglePbox[6]:=ultrasoundKnifeGripAngleIK(gripAngle); 
	m_gripAnglePbox[7]:=rot_x*kx;
	m_gripAnglePbox[8]:=rot_x*kx;
ELSE
	m_gripAnglePbox[7]:=rot_x*kx;
	m_gripAnglePbox[6]:=rot_y*ky;
	ra:=gripAngle;
	m_gripAnglePbox[4]:=rot_y*k13*kz+d*rot_z*kz+d*ra*kz/2;
	m_gripAnglePbox[5]:=-rot_y*k23*kz-d*rot_z*kz+d*ra*kz/2;
END_IF

// convert instrument joint position to motor joint position
o_jntPos[4] := m_gripAnglePbox[4] + m_jntPosOffset[4];
o_jntPos[5] := m_gripAnglePbox[5] + m_jntPosOffset[5];
o_jntPos[6] := m_gripAnglePbox[6] + m_jntPosOffset[6];
o_jntPos[7] := -m_gripAnglePbox[7] + m_jntPosOffset[7];
o_jntPos[8] := -m_gripAnglePbox[8] + m_jntPosOffset[8];
END_METHOD

// convert motor joint velocity to DH joint velocity
METHOD PUBLIC instruJntVelFK : BOOL
VAR_IN_OUT CONSTANT
	// motor joint velocity of slave arm
	i_jntVel :Vec8d;
END_VAR

VAR_IN_OUT
	// instrument DH  joint velocity
	r_DHJntVel :Vec6d;
END_VAR

VAR
	kx,ky,kz, k13, k23,openAngleDir:LREAL;
END_VAR
r_DHJntVel[1]:=i_jntVel[1];
r_DHJntVel[2]:=i_jntVel[2];
r_DHJntVel[3]:=i_jntVel[3];

// kinematic variables
openAngleDir:=-1;
kx:=-1;
ky:=m_instruTypeInfo.m_k2;
kz:=m_instruTypeInfo.m_k1;
k13:=m_instruTypeInfo.m_k3;
k23:=m_instruTypeInfo.m_k3;

r_DHJntVel[4]:=-i_jntVel[7]/kx;
r_DHJntVel[5]:=i_jntVel[6]/ky;
r_DHJntVel[6]:=(i_jntVel[4]-i_jntVel[5]-2*r_DHJntVel[5]*k13*kz)/(2*openAngleDir*kz);
r_DHJntVel[5]:=-r_DHJntVel[5];
r_DHJntVel[6]:=-r_DHJntVel[6];
END_METHOD

METHOD PROTECTED InstruSreiesFind : BOOL
VAR_INPUT
	i_NewValue:ULINT;
	i_ArrayData:ARRAY [1..100] OF ULINT;
	
END_VAR

VAR
	k1:INT;
END_VAR
InstruSreiesFind:=FALSE;
FOR k1:= 1 TO 100 BY 1 DO
	IF i_NewValue=i_ArrayData[k1] THEN
		InstruSreiesFind:=TRUE;
		EXIT;
	ELSE
		InstruSreiesFind:=FALSE;
	END_IF
END_FOR
END_METHOD

PROPERTY PUBLIC instruType : E_InstrumentType
GET
instruType := m_instruType;
END_GET
END_PROPERTY

PROPERTY instruTypeInfo :REFERENCE TO ST_InstruTypeInfo
GET
instruTypeInfo ref=m_instruTypeInfo;
END_GET
END_PROPERTY

PROPERTY nextScopePosture : E_EndoscopePosture
GET
nextScopePosture:= m_nextEndoscopePosture;
END_GET
SET
m_nextEndoscopePosture := nextScopePosture;
END_SET
END_PROPERTY

PROPERTY nextScopeType : E_EndoscopePosture
GET
nextScopeType:= m_nextEndoscopeType;
END_GET
SET
m_nextEndoscopeType := nextScopeType;
END_SET
END_PROPERTY

PROPERTY onChipData : REFERENCE TO ST_InstruOnChipData
GET
onChipData ref=m_onChipData;
END_GET
END_PROPERTY

METHOD PROTECTED proGrsapForcepsGripAngleFK : BOOL
VAR_INPUT
	frontAngle:LREAL;
END_VAR
VAR_OUTPUT
	endAngle:LREAL;
	Succeed:BOOL;
END_VAR
VAR
	// prograsp data
	AB :LREAL := 2.8;
	BC:LREAL := 5.26;
	initA:LREAL := 16.6 * g_deg2Rad; 
	initC:LREAL := 8.75*g_deg2Rad;
	
	SIN_C,Angle_Inc_C,Angle_C,Angle_A,Angle_Inc_A:LREAL;
END_VAR
//**************已知：器械前端开合角，求解：末端开合角***************//
// determine prograsp type data
IF InstruType_ProGraspForceps=m_instruType THEN
	AB:=g_proGraspAB;
	BC:=g_proGraspBC;
	initA := g_proGraspInitA;
	initC := g_proGraspInitC;
ELSIF InstruType_ForceBipolar=m_instruType THEN
	AB:=g_proGrasp2AB;
	BC:=g_proGrasp2BC;
	initA := g_proGrasp2InitA;
	initC := g_proGrasp2InitC;
END_IF

Angle_Inc_A:=frontAngle/2;
Angle_A:=initA+Angle_Inc_A;
Angle_A := LIMIT(0.0, Angle_A, pi);

SIN_C:=AB*SIN(Angle_A)/BC;
Angle_C:=ASIN(SIN_C);

Angle_Inc_C:=Angle_C-initC;
endAngle:=Angle_Inc_C*2;
END_METHOD

METHOD PROTECTED proGrsapForcepsGripAngleIK : BOOL
VAR_INPUT
	endAngle:LREAL;
END_VAR
VAR_OUTPUT
	frontAngle:LREAL;
	Succeed:BOOL;
END_VAR
VAR
	AB :LREAL := 2.8;
	BC:LREAL := 5.26;
	initA:LREAL := 16.6 * g_deg2Rad; 
	initC:LREAL := 8.75*g_deg2Rad;
	Angle_Inc_C,Angle_C,SIN_A,Angle_A,Angle_Inc_A:LREAL;
END_VAR
//***************已知：器械末端开合角，求解：前端开合角********************//
// determine prograsp type data
IF InstruType_ProGraspForceps=m_instruType THEN
	AB:=g_proGraspAB;
	BC:=g_proGraspBC;
	initA := g_proGraspInitA;
	initC := g_proGraspInitC;
ELSIF InstruType_ForceBipolar=m_instruType THEN
	AB:=g_proGrasp2AB;
	BC:=g_proGrasp2BC;
	initA := g_proGrasp2InitA;
	initC := g_proGrasp2InitC;
END_IF

Angle_Inc_C:=endAngle/2;
Angle_C:=initC+Angle_Inc_C;
Angle_C := LIMIT(0, Angle_C, pi);

SIN_A:=BC*SIN(Angle_C)/AB;
Angle_A:=ASIN(SIN_A);

Angle_Inc_A:=Angle_A-initA;
frontAngle:=Angle_Inc_A*2;
END_METHOD

METHOD PUBLIC readParameters : BOOL
VAR_INPUT
	startFlag :BOOL;
END_VAR

VAR
	paramIdx :INT;
	endoscopeData:UINT;
END_VAR
// TODO: read m_kinematic parameters from chip 
//Take the rising edge of the read signal
m_ReadDelay(IN:= m_Step=10, PT:= m_DealyTime, Q=> , ET=> );//计时器
IF startFlag AND m_curReadTries < m_maxReadTries THEN
	m_Step:=0;
	m_onChipData.m_InstruReadSucceed:=FALSE;
	m_onChipData.m_Error:=FALSE;
	m_onChipData.m_ErrorID:=0;
	m_resetArmLEDFlag :=TRUE;
END_IF


CASE m_Step OF
	
	0://向6093发送0x8000  0000---发送读取信号
		m_Value:=16#80000000; 
		m_SdoWrite(sNetId:= m_ArmNetId, nSlaveAddr:= m_JointInstruAddr, nSubIndex:= 0, nIndex:= 16#6093, pSrcBuf:= ADR(m_Value), cbBufLen:= SIZEOF(m_Value), bExecute:= TRUE, );
		IF NOT m_SdoWrite.bBusy THEN
			m_SdoWrite(bExecute:=FALSE);
			m_Step:=10;
		END_IF
		
		
	10://延时0.5s、防止值还没有返回
		IF m_ReadDelay.Q THEN
			m_Step:=20;
		END_IF

		
	20://从6093地址中拿值
		m_SdoRead(sNetId:= m_ArmNetId, nSlaveAddr:= m_JointInstruAddr,	nSubIndex:= 0, nIndex:= 16#6093, pDstBuf:= ADR(m_IDReadResult), cbBufLen:= SIZEOF(m_IDReadResult), bExecute:= TRUE, 	tTimeout:= , bBusy=> , bError=> , nErrId=> , cbRead=> );
		IF NOT m_SdoRead.bBusy THEN
			m_SdoRead(bExecute:=FALSE);
			m_Step:=30;
		END_IF	
		
	
	30://处理器械ID、低16位
		m_IDResult:=UDINT_TO_ULINT(16#0000FFFF AND m_IDReadResult);
		m_Step:=40;
		
		
	40://读取6095、器械序列号
		m_SdoRead(sNetId:= m_ArmNetId, nSlaveAddr:= m_JointInstruAddr,	nSubIndex:= 0, nIndex:= 16#6095, pDstBuf:= ADR(m_SeriesReadResult), cbBufLen:= SIZEOF(m_SeriesReadResult), bExecute:= TRUE, 	tTimeout:= , bBusy=> , bError=> , nErrId=> , cbRead=> );
		IF NOT m_SdoRead.bBusy THEN
			m_SdoRead(bExecute:=FALSE);
			m_Step:=50;
		END_IF	
	
		
	50://处理序列号，低30位
		m_onChipData.m_InstruseriesNum:=SHL(m_IDResult,31)+(16#7FFFFFFF AND m_SeriesReadResult);
		m_onChipData.m_InstruID:=LREAL_TO_INT(FLOOR(lr_in:= m_onChipData.m_InstruseriesNum/EXPT(10,9))); //取十进制前三位为器械ID
		IF m_onChipData.m_InstruID = InstruType_Endoscope THEN
			endoscopeData := LREAL_TO_UINT(FLOOR(lr_in:= m_onChipData.m_InstruseriesNum/EXPT(10,7)));
			endoscopeData := endoscopeData MOD 100;
			IF endoscopeData>= 25 THEN
				m_onChipData.m_InstruID := InstruType_NewEndoscope;
			END_IF
		END_IF
		m_Step:=60;
		
		
	60://读取6096---器械零点位置
		m_SdoRead(sNetId:= m_ArmNetId, nSlaveAddr:= m_JointInstruAddr,	nSubIndex:= 0, nIndex:= 16#6096, pDstBuf:= ADR(m_PosReadResult), cbBufLen:= SIZEOF(m_PosReadResult), bExecute:= TRUE, 	tTimeout:= , bBusy=> , bError=> , nErrId=> , cbRead=> );
		IF NOT m_SdoRead.bBusy THEN
			m_SdoRead(bExecute:=FALSE);
			m_Step:=70;
		END_IF	
		
		
	70: //处理位置，L1:0-9位，L2:10-19位，L3:20-29位
		zeroPosDecode(m_PosReadResult, o_q1=>m_onChipData.m_InstruPos[1],o_q2=>m_onChipData.m_InstruPos[2],o_q3=>m_onChipData.m_InstruPos[3]);
		m_onChipData.m_InstruPos[4] := m_jnt4ZeroPos;
		m_onChipData.m_InstruPos[5] := 0;
		
		m_Step:=80;
		
	80://读取器械使用次数 6094
		m_SdoRead(sNetId:= m_ArmNetId, nSlaveAddr:= m_JointInstruAddr,	nSubIndex:= 0, nIndex:= 16#6094, pDstBuf:= ADR(m_UsageReadResult), cbBufLen:= SIZEOF(m_UsageReadResult), bExecute:= TRUE, 	tTimeout:= , bBusy=> , bError=> , nErrId=> , cbRead=> );
		IF NOT m_SdoRead.bBusy THEN
			m_SdoRead(bExecute:=FALSE);
			m_Step:=90;
		END_IF	
		
		
	90://处理器械使用次数读取结果
		m_onChipData.m_InstruusageCounts:=m_UsageReadResult;
		m_InstruUsageToLED:=LIMIT(0,m_UsageReadResult,99);
		m_Step:=100;
		
		
	100://将器械使用次数写入LED
		m_Value:=ULINT_TO_UDINT(16#FFFF AND m_InstruUsageToLED) ;
		m_SdoWrite(sNetId:= m_ArmNetId, nSlaveAddr:= m_LEDAddr, nSubIndex:= 06, nIndex:= 16#6090, pSrcBuf:= ADR(m_Value), cbBufLen:= SIZEOF(m_Value), bExecute:= TRUE, tTimeout:= , bBusy=> , bError=> , nErrId=> );
		IF NOT m_SdoWrite.bBusy THEN
			m_SdoWrite(bExecute:=FALSE);
			m_Step:=110;
		END_IF
		
	110:
		// get insturment typeinfo
		m_onChipData.m_InstruReadSucceed:=checkInstruType();
		
		//结果诊断
		m_onChipData.m_ErrorID:=0;
		IF NOT(m_onChipData.m_InstruReadSucceed) THEN
			m_onChipData.m_Error:=TRUE;
			m_onChipData.m_ErrorID:=1;
			
		ELSIF SlaveArmControl.m_slaveRobot.m_endoscopeMounted AND m_instruType = InstruType_Endoscope THEN
			m_onChipData.m_InstruReadSucceed := FALSE;
			m_onChipData.m_Error:=TRUE;
			m_onChipData.m_ErrorID:=3;
			
//		ELSIF m_onChipData.m_InstruusageCounts>(m_instruTypeInfo.m_maxUseNum -1) AND m_instruType<>InstruType_Endoscope THEN
		ELSIF m_onChipData.m_InstruusageCounts>100 AND m_instruType<>InstruType_Endoscope THEN
			m_HaveRecord:=InstruSreiesFind(i_NewValue:=m_onChipData.m_InstruseriesNum , i_ArrayData:=GVL_interactUI.g_InstruSeriesRecord );
			IF m_HaveRecord THEN
				//
			ELSE
				m_onChipData.m_InstruReadSucceed := FALSE; 
				m_onChipData.m_Error:=TRUE;
				m_onChipData.m_ErrorID:=2;
			END_IF
		END_IF
		
		//处理当器械使用次数达到上限后、在同一场手术中还能使用
		IF m_onChipData.m_InstruReadSucceed AND m_onChipData.m_InstruusageCounts=(m_instruTypeInfo.m_maxUseNum -1) THEN		
			//TODO: check this part
			GVL_interactUI.g_InstruSeriesRecord:=InstruIDRecord(i_NewValue:= m_onChipData.m_InstruseriesNum, i_ArrayData:= GVL_interactUI.g_InstruSeriesRecord);
		END_IF
		
		m_Step :=-1;
		m_curReadTries := m_curReadTries +1;
	
END_CASE
END_METHOD

METHOD PUBLIC reset : BOOL
VAR_INPUT
END_VAR
VAR
	i:INT;
END_VAR
m_Step := -1;
m_curReadTries := 0;
m_onChipData.m_InstruID := 0;
m_onChipData.m_InstruseriesNum :=0;
m_onChipData.m_Error:=FALSE;
m_onChipData.m_ErrorID:=0;
m_onChipData.m_InstruReadSucceed:=FALSE;
m_instruType:=InstruType_UNKNOWM;

FOR i:= 4 TO 8 BY 1 DO
	m_jntPosOffset[i]:=0;
END_FOR

// init joint motion range
FOR i:=1 TO 3 DO
	m_wristMinDHJntPos[i]:=GVL_SlaveMotorParameters.g_minDHJntPos[i+3];
	m_wristMaxDHJntPos[i]:=GVL_SlaveMotorParameters.g_maxDHJntPos[i+3];
END_FOR

// reset endoscope type and posture
m_curEndoscopeType :=EndoScopeType_30;
m_nextEndoscopeType :=EndoScopeType_30;
m_curEndoscopePosture :=EndoscopePosture_HeadDown;
m_nextEndoscopePosture :=EndoscopePosture_HeadDown;

//arm LED reset
IF m_resetArmLEDFlag THEN
	m_Value:=0 ;
	m_SdoWrite(sNetId:= m_ArmNetId, nSlaveAddr:= m_LEDAddr, nSubIndex:= 06, nIndex:= 16#6090, pSrcBuf:= ADR(m_Value), cbBufLen:= SIZEOF(m_Value), bExecute:= TRUE, tTimeout:= , bBusy=> , bError=> , nErrId=> );
END_IF
IF NOT m_SdoWrite.bBusy THEN
	m_SdoWrite(bExecute:=FALSE);
	m_resetArmLEDFlag := FALSE;
END_IF
END_METHOD

PROPERTY resetArmLED : BOOL
SET
m_resetArmLEDFlag := resetArmLED;
END_SET
END_PROPERTY

METHOD ultrasoundKnifeGripAngleFK : LREAL
VAR_INPUT
	// motor joint position of slave arm
	i_jntPos :LREAL;
END_VAR

VAR
	m_jntPos : LREAL;
END_VAR
m_jntPos := i_jntPos;

m_jntPos := LIMIT (-20*g_deg2Rad,m_jntPos,70*g_deg2Rad);

ultrasoundKnifeGripAngleFK := ASIN((m_jntPos*g_uknifeMotorLead * g_uknifeLeverRatio/(2*pi) -  g_uknifeGripTravel * SIN(g_uknifeGripDividAngle))/g_uknifeGripTravel)+g_uknifeGripDividAngle;
END_METHOD

METHOD ultrasoundKnifeGripAngleIK : LREAL
VAR_INPUT
	// gripper angle
	i_gripAngle :LREAL;
END_VAR

VAR
	m_gripAngle : LREAL;
END_VAR
m_gripAngle := i_gripAngle;

ultrasoundKnifeGripAngleIK := (g_uknifeGripTravel * (SIN(g_uknifeGripDividAngle) - SIN(g_uknifeGripDividAngle - m_gripAngle))/(g_uknifeMotorLead*g_uknifeLeverRatio/(2*pi)));
END_METHOD

METHOD writeNumOfUseToChip : BOOL
VAR_INPUT
	startFlag :BOOL;
	i_useNumFromUI :UINT;
END_VAR
writeNumOfUseToChip := FALSE;
m_writeLDP(CLK:= startFlag, Q=> );
m_ReadNumDelay(IN:= m_useNumStep = 10, PT:= m_DealyTime, Q=> , ET=> );
IF m_writeLDP.Q THEN
	m_useNumStep:=0;
END_IF

CASE m_useNumStep OF
	0: 
		m_Value:=16#80000000; 
		m_SdoWrite(sNetId:= m_ArmNetId, nSlaveAddr:= m_JointInstruAddr, nSubIndex:= 0, nIndex:= 16#6094, pSrcBuf:= ADR(m_Value), cbBufLen:= SIZEOF(m_Value), bExecute:= TRUE, );
		IF NOT m_SdoWrite.bBusy THEN
			m_SdoWrite(bExecute:=FALSE);
			m_useNumStep:=10;
		END_IF
	
	10:
		IF m_ReadNumDelay.Q THEN
			m_useNumStep:=20;
		END_IF
		
	20:
		m_SdoRead(sNetId:= m_ArmNetId, nSlaveAddr:= m_JointInstruAddr,	nSubIndex:= 0, nIndex:= 16#6094, pDstBuf:= ADR(m_useNumReadResult), cbBufLen:= SIZEOF(m_useNumReadResult), bExecute:= TRUE, 	tTimeout:= , bBusy=> , bError=> , nErrId=> , cbRead=> );
		IF NOT m_SdoRead.bBusy THEN
			m_SdoRead(bExecute:=FALSE);
			m_useNumStep:=30;
		END_IF
		
	30://Verify the actual usage count and the usage count given by the UI
		IF m_useNumReadResult = i_useNumFromUI THEN
			m_useNumSendToLED := LIMIT(0, m_useNumReadResult, 99);
			m_useNumStep:=40;
		ELSE
			m_useNumStep:=50;
		END_IF
		
	40: 
		m_Value:=ULINT_TO_UDINT( m_useNumSendToLED) ;
		m_SdoWrite(sNetId:= m_ArmNetId, nSlaveAddr:= m_LEDAddr, nSubIndex:= 06, nIndex:= 16#6090, pSrcBuf:= ADR(m_Value), cbBufLen:= SIZEOF(m_Value), bExecute:= TRUE, tTimeout:= , bBusy=> , bError=> , nErrId=> );
		IF NOT m_SdoWrite.bBusy THEN
			m_SdoWrite(bExecute:=FALSE);
			m_onChipData.m_InstruUsageCounts:=m_useNumReadResult;
			writeNumOfUseToChip := TRUE;
			m_useNumStep:=-1;
		END_IF
		
END_CASE
END_METHOD

METHOD PUBLIC writeZeroPosToChip : BOOL
VAR_INPUT
	i_q1:LREAL;
	i_q2:LREAL;
	i_q3:LREAL;
END_VAR
zeroPosCode(i_q1,i_q2,i_q3, o_code=>m_zeroPosCode);

writeZeroPosToChip:=FALSE;
m_SdoWrite(sNetId:= m_ArmNetId, nSlaveAddr:= m_JointInstruAddr, nSubIndex:= 0, nIndex:= 16#6096, pSrcBuf:= ADR(m_zeroPosCode), cbBufLen:= SIZEOF(m_zeroPosCode), bExecute:= TRUE, );
IF NOT m_SdoWrite.bBusy THEN
	m_SdoWrite(bExecute:=FALSE);
	writeZeroPosToChip:=TRUE;
END_IF
END_METHOD

// code instrument joints(4/5/6) zero position as a UDINT
// joint1 : bit 21-30; joint2: bit 11-20; joint3: bit1-10
// zeroPos: [0, 2pi]; code:[0-3sFF]
METHOD PROTECTED zeroPosCode : BOOL
VAR_INPUT
	i_q1:LREAL;
	i_q2:LREAL;
	i_q3:LREAL;
END_VAR
VAR_OUTPUT
	o_code:UDINT;
END_VAR
VAR
	posCode:UDINT;
END_VAR
// highest bit set to 1
o_code:=2;

// joint1
posCode := LREAL_TO_UDINT(16#3FF * LIMIT(0,i_q1/g_2pi,1));
o_code := SHL(o_code, 10);
o_code := o_code OR posCode;

// joint2
posCode := LREAL_TO_UDINT(16#3FF * LIMIT(0,i_q2/g_2pi,1));
o_code := SHL(o_code, 10);
o_code := o_code OR posCode;

// joint3
posCode := LREAL_TO_UDINT(16#3FF * LIMIT(0,i_q3/g_2pi,1));
o_code := SHL(o_code, 10);
o_code := o_code OR posCode;
END_METHOD

// decode instrument joints(4/5/6) zero position from a UDINT
// joint1 : bit 21-30; joint2: bit 11-20; joint4: bit1-10
// zeroPos: [0, 2pi]; code:[0-2FF]
METHOD PROTECTED zeroPosDecode : BOOL
VAR_INPUT
	i_posCode :UDINT;
END_VAR
VAR_OUTPUT
	o_q1:LREAL;
	o_q2:LREAL;
	o_q3:LREAL;
END_VAR
VAR
	posCode:UDINT;
	ultraKnifePos : UDINT;
	posDir : UDINT;
END_VAR
// ultrasound knife 
IF (InstruType_UltrasoundKnifeS = m_onChipData.m_InstruID OR InstruType_UltrasoundKnifeU = m_onChipData.m_InstruID) THEN
	ultraKnifePos := i_posCode;
	posCode := i_posCode AND 16#FFFFF;
	posDir := SHR(ultraKnifePos,20);
	IF posDir = 0 THEN
		o_q3 := (UDINT_TO_LREAL(posCode)/1000);
	ELSIF posDir = 1 THEN
		o_q3 := g_2pi - (UDINT_TO_LREAL(posCode)/1000);
	END_IF
ELSE
	
	// joint3
	posCode := i_posCode AND 16#3FF;
	o_q3 := g_2pi *  posCode/16#3FF;
	
	// joint2
	i_posCode := SHR(i_posCode, 10);
	posCode := i_posCode AND 16#3FF;
	o_q2 := g_2pi *  posCode/16#3FF;
	
	// joint1
	i_posCode := SHR(i_posCode, 10);
	posCode := i_posCode AND 16#3FF;
	o_q1 := g_2pi *  posCode/16#3FF;
END_IF
END_METHOD

END_FUNCTION_BLOCK

// ---- FBs_SlaveControllers/FB_SlaveCtrlError.TcPOU
// Brief: Slave Arm Error Hold
FUNCTION_BLOCK PUBLIC FB_SlaveCtrlError EXTENDS FB_SlaveArmCtrlBase
VAR
END_VAR

// override this function in each exact controller
METHOD PROTECTED calcCmdJntPos : BOOL
VAR_IN_OUT CONSTANT
	// endoscope pose in cart coordinate
	i_endoscopePose : ST_Frame;
	
	// master arm data
	i_masterStatus :ST_MasterStatus;
	
	// setup arm data
	i_setupStatus: ST_SetupStatus;
	
	// slave arm data
	i_slaveArm :FB_SlaveArm;
END_VAR
m_cmdJntPos := i_slaveArm.curJntPos;
END_METHOD

// override this function in each exact controller
// NOTICE: set joint control mode here, and do some initialization if needed
METHOD PUBLIC init : BOOL
VAR_IN_OUT CONSTANT
	i_slaveArm	:FB_SlaveArm;
END_VAR
VAR_IN_OUT 
	r_slaveArmCtrlCmd :ST_SlaveArmCtrlCmds;
END_VAR


VAR
	i:INT;
END_VAR
SUPER^.Init(i_slaveArm,r_slaveArmCtrlCmd);

// disable first three joints
m_jntEnableFlag[1]:= 0;
m_jntEnableFlag[2]:= 0;
m_jntEnableFlag[3]:= 0;

// disable instrument joints which is in error 
FOR i:=4 TO g_sJntNum DO
	IF SafetyCheck.m_SafetyCheck.m_jntErrFlag[i_slaveArm.armIdx, i+g_setupJntNum, 2] OR  SafetyCheck.m_SafetyCheck.m_jntErrFlag[i_slaveArm.armIdx, i+g_setupJntNum, 3] 
		OR SafetyCheck.m_SafetyCheck.m_jntErrFlag[i_slaveArm.armIdx, 0, 3] OR NOT SlaveArmControl.m_slaveRobot.m_selfCheckPass[i_slaveArm.armIdx]  THEN
		m_jntEnableFlag[i] := 0;
	ELSE
		m_jntEnableFlag[i] := 1;
	END_IF
	IF SafetyCheck.m_SafetyCheck.m_jntErrFlag[i_slaveArm.armIdx, 0, 2] AND (i =4 OR  i= 5) THEN
		m_jntEnableFlag[i] := 0;
	END_IF
END_FOR
 
 // update commands to arm
copyCmds(r_slaveArmCtrlCmd);
END_METHOD

END_FUNCTION_BLOCK

// ---- FBs_SlaveControllers/FB_SlaveArmCtrlBase.TcPOU
// Slave Arm Base Controller, Hold at Current Posture
FUNCTION_BLOCK FB_SlaveArmCtrlBase IMPLEMENTS I_SlaveArmCtrl
VAR_INPUT
END_VAR
VAR_OUTPUT
END_VAR
VAR
	// flag if the controller has finished all its jobs
	m_isFinished:BOOL:=FALSE;
	
	// controller execute time period
	m_timePeriod :LREAL:=0;
	
	// flag to hold last commands
	m_holdLastCmds :BOOL := FALSE;
	
	// arm control data
	// NOTE: simulated joint position is usd for kinematic controller 
	//		while command joint position is used for real robot controller
	// 		They are identical for the most time, but in some cases, simulated position is filted to get command one 
	m_simJntPos :Vec8d; 
	m_cmdJntPos : VEC8d; 
	m_cmdJntVel : VEC8d;
	m_cmdJntAcc : VEC8d;
	m_cmdJntTrq : VEC8d;
	m_jntOPMode : Vec8i;
	m_jntEnableFlag :Vec8i;
	m_cmdCartPose : ST_Frame;
	m_cmdCartTwist : Vec6d;
	m_FFJntTrq :Vec8d;
	
END_VAR

// override this function in each exact controller
METHOD PROTECTED calcCmdJntPos : BOOL
VAR_IN_OUT CONSTANT
	// endoscope pose in cart coordinate
	i_endoscopePose : ST_Frame;
	
	// master arm data
	i_masterStatus :ST_MasterStatus;
	
	// setup arm data
	i_setupStatus: ST_SetupStatus;
	
	// slave arm data
	i_slaveArm :FB_SlaveArm;
END_VAR
IF isFinished THEN
	RETURN;
END_IF
END_METHOD

// override this function in each exact controller
METHOD PROTECTED calcCmdJntTrq : BOOL
VAR_IN_OUT CONSTANT
	// endoscope pose in cart coordinate
	i_endoscopePose : ST_Frame;
	
	// master arm data
	i_masterStatus :ST_MasterStatus;
	
	// setup arm data
	i_setupStatus: ST_SetupStatus;
	
	// slave arm data
	i_slaveArm :FB_SlaveArm;
END_VAR
IF isFinished THEN
	RETURN;
END_IF
END_METHOD

METHOD checkToHoldLastCmds : BOOL
VAR_IN_OUT CONSTANT
	i_slaveArm :FB_SlaveArm;
END_VAR
VAR
	j:INT;
	maxJntErr:LREAL;
	jntCtrlErr:Vec8d;
END_VAR
// check if to hold the command joint position unchanged
vecSub(i_slaveArm.m_cmdJntPos, i_slaveArm.m_curJntPos,jntCtrlErr);
maxJntErr:=0.0;
FOR j:=1 TO g_sJntNum DO
	maxJntErr:= MAX(maxJntErr, ABS(jntCtrlErr[j]));
END_FOR

checkToHoldLastCmds := (maxJntErr<GVL_SlaveControlParameters.g_jntCtrlErrForCmdHold);
END_METHOD

